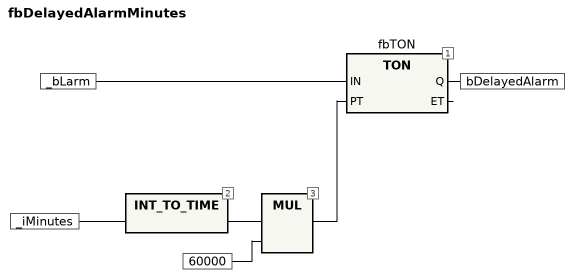
_CFC_ (* Continuous Function Chart, elements in execution order *)
#0 bDelayedAlarm <= #1.Q
#1 fbTON:TON(IN: _bLarm, PT: #3)
#2 INT_TO_TIME(_iMinutes)
#3 MUL(#2, 60000)
_END_CFC_
(* the same logic as Structured Text *)
bDelayedAlarm := fbTON.Q;
fbTON(IN := _bLarm, PT := _t13);
_t13 := INT_TO_TIME(_iMinutes) * 60000;
END_FUNCTION_BLOCK

(* POU xRIO_komfel/RIO_COM_L, CFC *)
PROGRAM RIO_COM_L
VAR

	State1 AT%I*:UINT;			(* Kommunikationsfel RIO1 *)
	State2 AT%I*:UINT;			(* Kommunikationsfel RIO2 *)
	State3 AT%I*:UINT;			(* Kommunikationsfel RIO3 *)
	State4 AT%I*:UINT;			(* Kommunikationsfel RIO4 *)
	State5 AT%I*:UINT;			(* Kommunikationsfel RIO5 *)

	KBusState1 AT%I*:UINT;			(* KBus/IO-fel  RIO1 *)
	KBusState2 AT%I*:UINT;			(* KBus/IO-fel  RIO2 *)
	KBusState3 AT%I*:UINT;			(* KBus/IO-fel  RIO3 *)
	KBusState4 AT%I*:UINT;			(* KBus/IO-fel  RIO4 *)
	KBusState5 AT%I*:UINT;			(* KBus/IO-fel  RIO5 *)

	Komfel1:BOOL;
	Komfel2:BOOL;
	Komfel3:BOOL;
	Komfel4:BOOL;
	Komfel5:BOOL;

	KBusfel1	:BOOL;
	KBusfel2	:BOOL;
	KBusfel3	:BOOL;
	KBusfel4	:BOOL;
	KBusfel5	:BOOL;

	KOMFELDELAY1: TON;
	KOMFELDELAY2: TON;
	KOMFELDELAY3: TON;
	KOMFELDELAY4: TON;
	KOMFELDELAY5: TON;
	IODELAY1: TON;
	IODELAY2: TON;
	IODELAY3: TON;
	IODELAY4: TON;
	IODELAY5: TON;
END_VAR
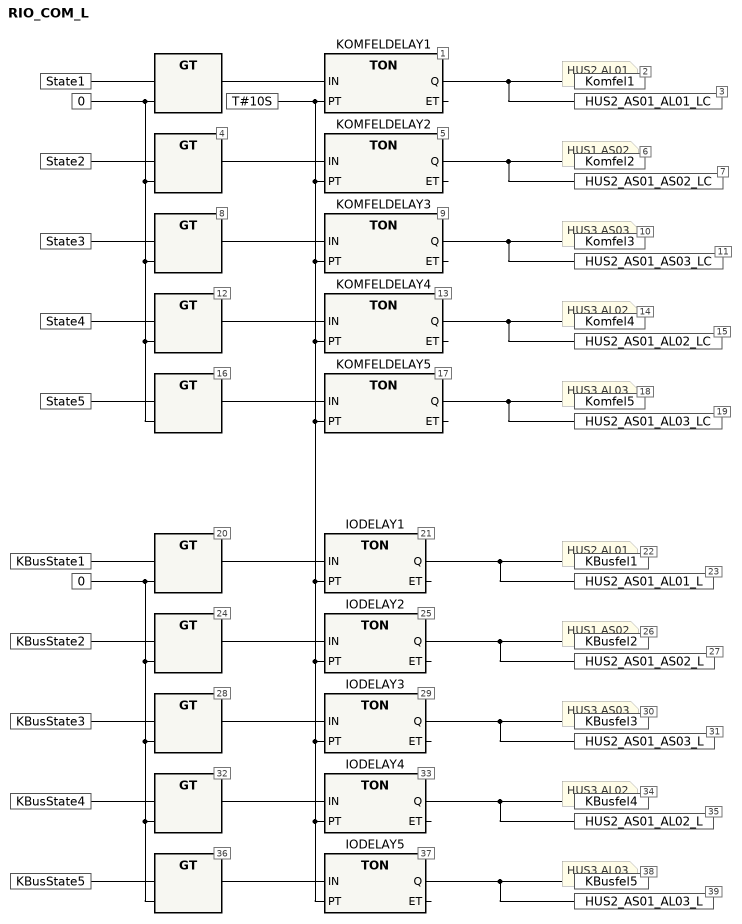
_CFC_ (* Continuous Function Chart, elements in execution order *)
(* HUS3 AL03 *)
(* HUS1 AS02 *)
(* HUS3 AL02 *)
(* HUS3 AS03 *)
(* HUS2 AL01 *)
(* HUS3 AL03 *)
(* HUS1 AS02 *)
(* HUS3 AL02 *)
(* HUS3 AS03 *)
(* HUS2 AL01 *)
#0 GT(State1, 0)
#1 KOMFELDELAY1:TON(IN: #0, PT: T#10S)
#2 Komfel1 <= #1.Q
#3 HUS2_AS01_AL01_LC <= #1.Q
#4 GT(State2, 0)
#5 KOMFELDELAY2:TON(IN: #4, PT: T#10S)
#6 Komfel2 <= #5.Q
#7 HUS2_AS01_AS02_LC <= #5.Q
#8 GT(State3, 0)
#9 KOMFELDELAY3:TON(IN: #8, PT: T#10S)
#10 Komfel3 <= #9.Q
#11 HUS2_AS01_AS03_LC <= #9.Q
#12 GT(State4, 0)
#13 KOMFELDELAY4:TON(IN: #12, PT: T#10S)
#14 Komfel4 <= #13.Q
#15 HUS2_AS01_AL02_LC <= #13.Q
#16 GT(State5, 0)
#17 KOMFELDELAY5:TON(IN: #16, PT: T#10S)
#18 Komfel5 <= #17.Q
#19 HUS2_AS01_AL03_LC <= #17.Q
#20 GT(KBusState1, 0)
#21 IODELAY1:TON(IN: #20, PT: T#10S)
#22 KBusfel1 <= #21.Q
#23 HUS2_AS01_AL01_L <= #21.Q
#24 GT(KBusState2, 0)
#25 IODELAY2:TON(IN: #24, PT: T#10S)
#26 KBusfel2 <= #25.Q
#27 HUS2_AS01_AS02_L <= #25.Q
#28 GT(KBusState3, 0)
#29 IODELAY3:TON(IN: #28, PT: T#10S)
#30 KBusfel3 <= #29.Q
#31 HUS2_AS01_AS03_L <= #29.Q
#32 GT(KBusState4, 0)
#33 IODELAY4:TON(IN: #32, PT: T#10S)
#34 KBusfel4 <= #33.Q
#35 HUS2_AS01_AL02_L <= #33.Q
#36 GT(KBusState5, 0)
#37 IODELAY5:TON(IN: #36, PT: T#10S)
#38 KBusfel5 <= #37.Q
#39 HUS2_AS01_AL03_L <= #37.Q
_END_CFC_
(* the same logic as Structured Text *)
(* HUS3 AL03 *)
(* HUS1 AS02 *)
(* HUS3 AL02 *)
(* HUS3 AS03 *)
(* HUS2 AL01 *)
(* HUS3 AL03 *)
(* HUS1 AS02 *)
(* HUS3 AL02 *)
(* HUS3 AS03 *)
(* HUS2 AL01 *)
KOMFELDELAY1(IN := State1 > 0, PT := T#10S);
Komfel1 := KOMFELDELAY1.Q;
HUS2_AS01_AL01_LC := KOMFELDELAY1.Q;
KOMFELDELAY2(IN := State2 > 0, PT := T#10S);
Komfel2 := KOMFELDELAY2.Q;
HUS2_AS01_AS02_LC := KOMFELDELAY2.Q;
KOMFELDELAY3(IN := State3 > 0, PT := T#10S);
Komfel3 := KOMFELDELAY3.Q;
HUS2_AS01_AS03_LC := KOMFELDELAY3.Q;
KOMFELDELAY4(IN := State4 > 0, PT := T#10S);
Komfel4 := KOMFELDELAY4.Q;
HUS2_AS01_AL02_LC := KOMFELDELAY4.Q;
KOMFELDELAY5(IN := State5 > 0, PT := T#10S);
Komfel5 := KOMFELDELAY5.Q;
HUS2_AS01_AL03_LC := KOMFELDELAY5.Q;
IODELAY1(IN := KBusState1 > 0, PT := T#10S);
KBusfel1 := IODELAY1.Q;
HUS2_AS01_AL01_L := IODELAY1.Q;
IODELAY2(IN := KBusState2 > 0, PT := T#10S);
KBusfel2 := IODELAY2.Q;
HUS2_AS01_AS02_L := IODELAY2.Q;
IODELAY3(IN := KBusState3 > 0, PT := T#10S);
KBusfel3 := IODELAY3.Q;
HUS2_AS01_AS03_L := IODELAY3.Q;
IODELAY4(IN := KBusState4 > 0, PT := T#10S);
KBusfel4 := IODELAY4.Q;
HUS2_AS01_AL02_L := IODELAY4.Q;
IODELAY5(IN := KBusState5 > 0, PT := T#10S);
KBusfel5 := IODELAY5.Q;
HUS2_AS01_AL03_L := IODELAY5.Q;
END_PROGRAM

(* POU _IOs_Uppdelat_per_skåp/HUS1_AS02/_IO/HUS1_AS02_IO_MAIN, CFC *)
PROGRAM HUS1_AS02_IO_MAIN
VAR
END_VAR
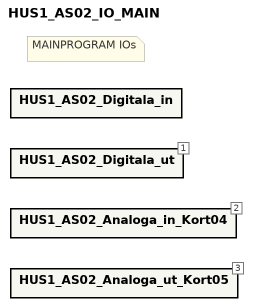
_CFC_ (* Continuous Function Chart, elements in execution order *)
(* MAINPROGRAM IOs *)
#0 HUS1_AS02_Digitala_in()
#1 HUS1_AS02_Digitala_ut()
#2 HUS1_AS02_Analoga_in_Kort04()
#3 HUS1_AS02_Analoga_ut_Kort05()
_END_CFC_
(* the same logic as Structured Text *)
(* MAINPROGRAM IOs *)
HUS1_AS02_Digitala_in();
HUS1_AS02_Digitala_ut();
HUS1_AS02_Analoga_in_Kort04();
HUS1_AS02_Analoga_ut_Kort05();
END_PROGRAM

(* POU _IOs_Uppdelat_per_skåp/HUS1_AS02/_IO/HUS1_AS02_Digitala_in, CFC *)
PROGRAM HUS1_AS02_Digitala_in

VAR


END_VAR
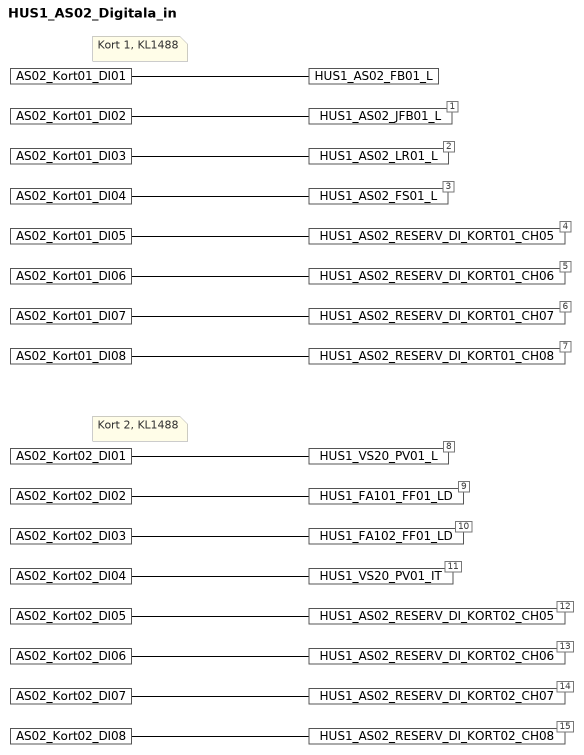
_CFC_ (* Continuous Function Chart, elements in execution order *)
(* Kort 1, KL1488 *)
(* Kort 2, KL1488 *)
#0 HUS1_AS02_FB01_L <= AS02_Kort01_DI01
#1 HUS1_AS02_JFB01_L <= AS02_Kort01_DI02
#2 HUS1_AS02_LR01_L <= AS02_Kort01_DI03
#3 HUS1_AS02_FS01_L <= AS02_Kort01_DI04
#4 HUS1_AS02_RESERV_DI_KORT01_CH05 <= AS02_Kort01_DI05
#5 HUS1_AS02_RESERV_DI_KORT01_CH06 <= AS02_Kort01_DI06
#6 HUS1_AS02_RESERV_DI_KORT01_CH07 <= AS02_Kort01_DI07
#7 HUS1_AS02_RESERV_DI_KORT01_CH08 <= AS02_Kort01_DI08
#8 HUS1_VS20_PV01_L <= AS02_Kort02_DI01
#9 HUS1_FA101_FF01_LD <= AS02_Kort02_DI02
#10 HUS1_FA102_FF01_LD <= AS02_Kort02_DI03
#11 HUS1_VS20_PV01_IT <= AS02_Kort02_DI04
#12 HUS1_AS02_RESERV_DI_KORT02_CH05 <= AS02_Kort02_DI05
#13 HUS1_AS02_RESERV_DI_KORT02_CH06 <= AS02_Kort02_DI06
#14 HUS1_AS02_RESERV_DI_KORT02_CH07 <= AS02_Kort02_DI07
#15 HUS1_AS02_RESERV_DI_KORT02_CH08 <= AS02_Kort02_DI08
_END_CFC_
(* the same logic as Structured Text *)
(* Kort 1, KL1488 *)
(* Kort 2, KL1488 *)
HUS1_AS02_FB01_L := AS02_Kort01_DI01;
HUS1_AS02_JFB01_L := AS02_Kort01_DI02;
HUS1_AS02_LR01_L := AS02_Kort01_DI03;
HUS1_AS02_FS01_L := AS02_Kort01_DI04;
HUS1_AS02_RESERV_DI_KORT01_CH05 := AS02_Kort01_DI05;
HUS1_AS02_RESERV_DI_KORT01_CH06 := AS02_Kort01_DI06;
HUS1_AS02_RESERV_DI_KORT01_CH07 := AS02_Kort01_DI07;
HUS1_AS02_RESERV_DI_KORT01_CH08 := AS02_Kort01_DI08;
HUS1_VS20_PV01_L := AS02_Kort02_DI01;
HUS1_FA101_FF01_LD := AS02_Kort02_DI02;
HUS1_FA102_FF01_LD := AS02_Kort02_DI03;
HUS1_VS20_PV01_IT := AS02_Kort02_DI04;
HUS1_AS02_RESERV_DI_KORT02_CH05 := AS02_Kort02_DI05;
HUS1_AS02_RESERV_DI_KORT02_CH06 := AS02_Kort02_DI06;
HUS1_AS02_RESERV_DI_KORT02_CH07 := AS02_Kort02_DI07;
HUS1_AS02_RESERV_DI_KORT02_CH08 := AS02_Kort02_DI08;
END_PROGRAM

(* POU _IOs_Uppdelat_per_skåp/HUS1_AS02/_IO/HUS1_AS02_Digitala_ut, CFC *)
PROGRAM HUS1_AS02_Digitala_ut


VAR
	HUS1_Kort03_DU01: BOOL;
	HUS1_Kort03_DU02: BOOL;
	HUS1_Kort03_DU03: BOOL;
	HUS1_HUS1_RESERV_DU_KORT03_CH04: BOOL;
	HUS1_Kort03_DU04: BOOL;
END_VAR
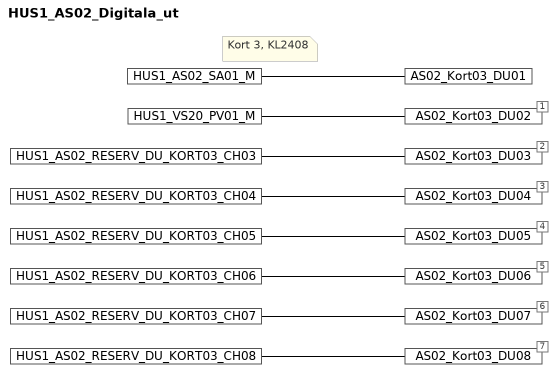
_CFC_ (* Continuous Function Chart, elements in execution order *)
(* Kort 3, KL2408 *)
#0 AS02_Kort03_DU01 <= HUS1_AS02_SA01_M
#1 AS02_Kort03_DU02 <= HUS1_VS20_PV01_M
#2 AS02_Kort03_DU03 <= HUS1_AS02_RESERV_DU_KORT03_CH03
#3 AS02_Kort03_DU04 <= HUS1_AS02_RESERV_DU_KORT03_CH04
#4 AS02_Kort03_DU05 <= HUS1_AS02_RESERV_DU_KORT03_CH05
#5 AS02_Kort03_DU06 <= HUS1_AS02_RESERV_DU_KORT03_CH06
#6 AS02_Kort03_DU07 <= HUS1_AS02_RESERV_DU_KORT03_CH07
#7 AS02_Kort03_DU08 <= HUS1_AS02_RESERV_DU_KORT03_CH08
_END_CFC_
(* the same logic as Structured Text *)
(* Kort 3, KL2408 *)
AS02_Kort03_DU01 := HUS1_AS02_SA01_M;
AS02_Kort03_DU02 := HUS1_VS20_PV01_M;
AS02_Kort03_DU03 := HUS1_AS02_RESERV_DU_KORT03_CH03;
AS02_Kort03_DU04 := HUS1_AS02_RESERV_DU_KORT03_CH04;
AS02_Kort03_DU05 := HUS1_AS02_RESERV_DU_KORT03_CH05;
AS02_Kort03_DU06 := HUS1_AS02_RESERV_DU_KORT03_CH06;
AS02_Kort03_DU07 := HUS1_AS02_RESERV_DU_KORT03_CH07;
AS02_Kort03_DU08 := HUS1_AS02_RESERV_DU_KORT03_CH08;
END_PROGRAM

(* POU _IOs_Uppdelat_per_skåp/HUS1_AS02/_IO/ANALOGA IN/Kort04/HUS1_AS02_Analoga_in_Kort04, CFC *)
PROGRAM HUS1_AS02_Analoga_in_Kort04
VAR
	bLG01: BOOL;
	bLG02: BOOL;
	bLG03: BOOL;
	bLG04: BOOL;
	bLG05: BOOL;
	bLG06: BOOL;
	bLG07: BOOL;
	bLG08: BOOL;

(*TEMP*)
	FT1:INT;
	LG_FL1:INT;
	FT2:INT;
	LG_FL2:INT;
	FT3:INT;
	LG_FL3:INT;
	FT4:INT;
	LG_FL4:INT;
	FT5:INT;
	LG_FL5:INT;
	FT6:INT;
	LG_FL6:INT;
	FT7:INT;
	LG_FL7:INT;
	FT8:INT;
	LG_FL8:INT;

END_VAR
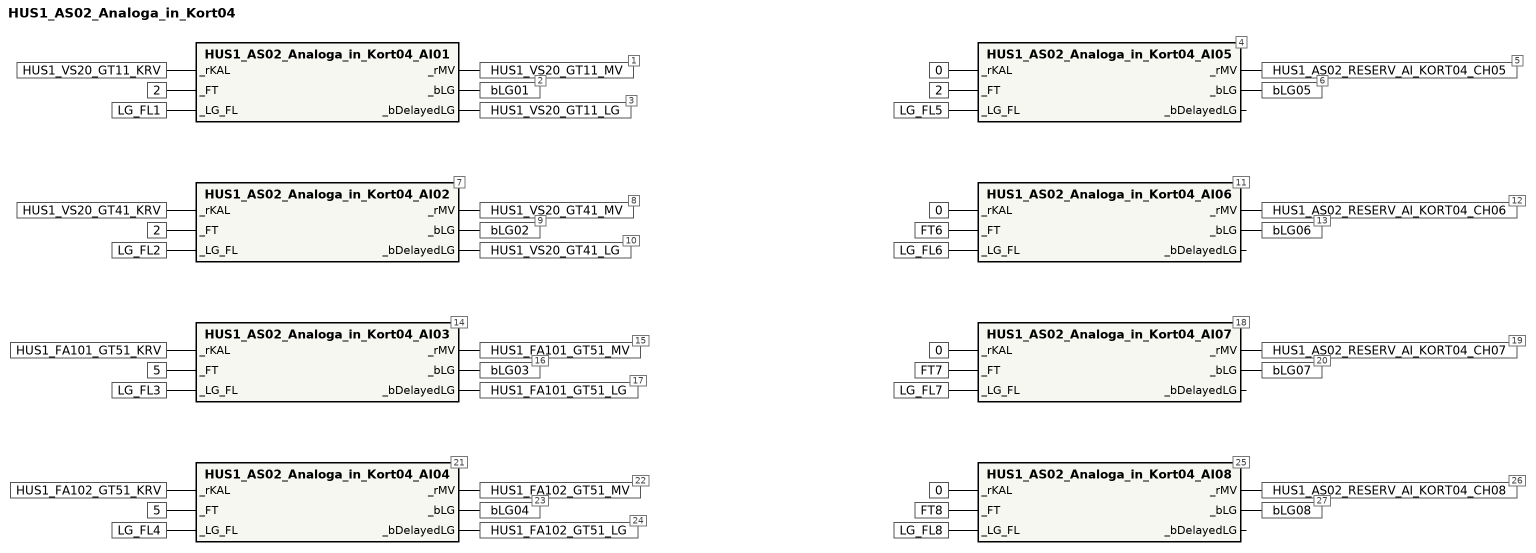
_CFC_ (* Continuous Function Chart, elements in execution order *)
#0 HUS1_AS02_Analoga_in_Kort04_AI01(_rKAL: HUS1_VS20_GT11_KRV, _FT: 2, _LG_FL: LG_FL1)
#1 HUS1_VS20_GT11_MV <= #0._rMV
#2 bLG01 <= #0._bLG
#3 HUS1_VS20_GT11_LG <= #0._bDelayedLG
#4 HUS1_AS02_Analoga_in_Kort04_AI05(_rKAL: 0, _FT: 2, _LG_FL: LG_FL5)
#5 HUS1_AS02_RESERV_AI_KORT04_CH05 <= #4._rMV
#6 bLG05 <= #4._bLG
#7 HUS1_AS02_Analoga_in_Kort04_AI02(_rKAL: HUS1_VS20_GT41_KRV, _FT: 2, _LG_FL: LG_FL2)
#8 HUS1_VS20_GT41_MV <= #7._rMV
#9 bLG02 <= #7._bLG
#10 HUS1_VS20_GT41_LG <= #7._bDelayedLG
#11 HUS1_AS02_Analoga_in_Kort04_AI06(_rKAL: 0, _FT: FT6, _LG_FL: LG_FL6)
#12 HUS1_AS02_RESERV_AI_KORT04_CH06 <= #11._rMV
#13 bLG06 <= #11._bLG
#14 HUS1_AS02_Analoga_in_Kort04_AI03(_rKAL: HUS1_FA101_GT51_KRV, _FT: 5, _LG_FL: LG_FL3)
#15 HUS1_FA101_GT51_MV <= #14._rMV
#16 bLG03 <= #14._bLG
#17 HUS1_FA101_GT51_LG <= #14._bDelayedLG
#18 HUS1_AS02_Analoga_in_Kort04_AI07(_rKAL: 0, _FT: FT7, _LG_FL: LG_FL7)
#19 HUS1_AS02_RESERV_AI_KORT04_CH07 <= #18._rMV
#20 bLG07 <= #18._bLG
#21 HUS1_AS02_Analoga_in_Kort04_AI04(_rKAL: HUS1_FA102_GT51_KRV, _FT: 5, _LG_FL: LG_FL4)
#22 HUS1_FA102_GT51_MV <= #21._rMV
#23 bLG04 <= #21._bLG
#24 HUS1_FA102_GT51_LG <= #21._bDelayedLG
#25 HUS1_AS02_Analoga_in_Kort04_AI08(_rKAL: 0, _FT: FT8, _LG_FL: LG_FL8)
#26 HUS1_AS02_RESERV_AI_KORT04_CH08 <= #25._rMV
#27 bLG08 <= #25._bLG
_END_CFC_
(* the same logic as Structured Text *)
HUS1_AS02_Analoga_in_Kort04_AI01(_rKAL := HUS1_VS20_GT11_KRV, _FT := 2, _LG_FL := LG_FL1);
HUS1_VS20_GT11_MV := HUS1_AS02_Analoga_in_Kort04_AI01._rMV;
bLG01 := HUS1_AS02_Analoga_in_Kort04_AI01._bLG;
HUS1_VS20_GT11_LG := HUS1_AS02_Analoga_in_Kort04_AI01._bDelayedLG;
HUS1_AS02_Analoga_in_Kort04_AI05(_rKAL := 0, _FT := 2, _LG_FL := LG_FL5);
HUS1_AS02_RESERV_AI_KORT04_CH05 := HUS1_AS02_Analoga_in_Kort04_AI05._rMV;
bLG05 := HUS1_AS02_Analoga_in_Kort04_AI05._bLG;
HUS1_AS02_Analoga_in_Kort04_AI02(_rKAL := HUS1_VS20_GT41_KRV, _FT := 2, _LG_FL := LG_FL2);
HUS1_VS20_GT41_MV := HUS1_AS02_Analoga_in_Kort04_AI02._rMV;
bLG02 := HUS1_AS02_Analoga_in_Kort04_AI02._bLG;
HUS1_VS20_GT41_LG := HUS1_AS02_Analoga_in_Kort04_AI02._bDelayedLG;
HUS1_AS02_Analoga_in_Kort04_AI06(_rKAL := 0, _FT := FT6, _LG_FL := LG_FL6);
HUS1_AS02_RESERV_AI_KORT04_CH06 := HUS1_AS02_Analoga_in_Kort04_AI06._rMV;
bLG06 := HUS1_AS02_Analoga_in_Kort04_AI06._bLG;
HUS1_AS02_Analoga_in_Kort04_AI03(_rKAL := HUS1_FA101_GT51_KRV, _FT := 5, _LG_FL := LG_FL3);
HUS1_FA101_GT51_MV := HUS1_AS02_Analoga_in_Kort04_AI03._rMV;
bLG03 := HUS1_AS02_Analoga_in_Kort04_AI03._bLG;
HUS1_FA101_GT51_LG := HUS1_AS02_Analoga_in_Kort04_AI03._bDelayedLG;
HUS1_AS02_Analoga_in_Kort04_AI07(_rKAL := 0, _FT := FT7, _LG_FL := LG_FL7);
HUS1_AS02_RESERV_AI_KORT04_CH07 := HUS1_AS02_Analoga_in_Kort04_AI07._rMV;
bLG07 := HUS1_AS02_Analoga_in_Kort04_AI07._bLG;
HUS1_AS02_Analoga_in_Kort04_AI04(_rKAL := HUS1_FA102_GT51_KRV, _FT := 5, _LG_FL := LG_FL4);
HUS1_FA102_GT51_MV := HUS1_AS02_Analoga_in_Kort04_AI04._rMV;
bLG04 := HUS1_AS02_Analoga_in_Kort04_AI04._bLG;
HUS1_FA102_GT51_LG := HUS1_AS02_Analoga_in_Kort04_AI04._bDelayedLG;
HUS1_AS02_Analoga_in_Kort04_AI08(_rKAL := 0, _FT := FT8, _LG_FL := LG_FL8);
HUS1_AS02_RESERV_AI_KORT04_CH08 := HUS1_AS02_Analoga_in_Kort04_AI08._rMV;
bLG08 := HUS1_AS02_Analoga_in_Kort04_AI08._bLG;
END_PROGRAM

(* POU _IOs_Uppdelat_per_skåp/HUS1_AS02/_IO/ANALOGA IN/Kort04/HUS1_AS02_Analoga_in_Kort04_AI01, FAI *)
PROGRAM HUS1_AS02_Analoga_in_Kort04_AI01
(*#####################################   Temperature Sensor Ex2   ################################################################*)
VAR
	(*===========================Configuration of terminal==========================================*)
	fbConfigureKL32xx					:FB_HVACConfigureKL32xx;
	_byCtrlKL32xx                         			AT %Q*: BYTE;
	_iDataOutKL32xx                       		AT %Q*: INT;
	_iDataInKL32xx 					AT%I*:INT;(* Raw Value from the Terminal *)
	_byStatusKL32xx 			AT%I*:BYTE;(* Statusbyte from Terminal *)

	_bScanSensor              					: BOOL;
	_tTimeOut                 					: TIME := T#5s;
	_bSetSensor               					: BOOL;
	bReady                               				: BOOL;
	byOutStatus                          			: BYTE;
	iOutDataIn                           				: INT;
	_eBusTerminalKL32xx                   		: E_HVACBusTerminal_KL32xx;
	_eStatusScanSensorType                	: E_HVACSensorType;
	_bErrorGeneral                        			: BOOL;
	_byError                              				: BYTE;
	_bErrorCommunication                  		: BOOL;
	_bErrorBusTerminalNotSupported   	: BOOL;
	_bErrorSensorType                     		: BOOL;
	_bErrorScanSensor                     		: BOOL;
	(*========================================================================================*)

	_bReset_Local					:BOOL;
	_bSetDefaultTempSens			:BOOL;

	(*========================================================================================*)
	FBHVACTemperatureSensor: FB_HVACTemperatureSensor;
	eDataSecurityType					: E_HVACDataSecurityType:=1;
	bSetDefault								:BOOL;
	iRawValue								:INT;
	byStatusRawValue						:BYTE;
	bEnableLimitCtrl							:BOOL;
	bReset									:BOOL;
	bErrorGeneral					:BOOL;
	byError							:BYTE;
	bErrorShortCircuit				:BOOL;
	bErrorBrokenSensor				:BOOL;
	bErrorHighLimit					:BOOL;
	bErrorLowLimit					:BOOL;
	bErrorCycleTime					:BOOL;
	bInvalidParameter				:BOOL;
	rOffset									:REAL;
	rHighLimit								:REAL;
	rLowLimit								:REAL;
	rReplacementValue						:REAL;
	tFilterTime								:TIME;
	eTemperatureSensorMode				:E_HVACTemperatureSensorMode:=2;
	fbAlarmD: fbDelayedAlarmMinutes;

END_VAR

VAR_INPUT
	_rKAL						: REAL;	(*Kalibrering*)
	_FT						:INT;		(*Filtertid*)
	_LG_FL					:INT;		(* Larmfördröjning givarfel *)
END_VAR

VAR_OUTPUT
	_rMV						:REAL;		(* Mätvärde *)
	_bLG						:BOOL; 	(*Givarfel*)
	_bDelayedLG				:BOOL;	(* Fördröjt givarfel *)
END_VAR
(* body not read: cfc101 *)
END_PROGRAM

(* POU _IOs_Uppdelat_per_skåp/HUS1_AS02/_IO/ANALOGA IN/Kort04/HUS1_AS02_Analoga_in_Kort04_AI05, FAI *)
PROGRAM HUS1_AS02_Analoga_in_Kort04_AI05
(*#####################################   Temperature Sensor Ex2   ################################################################*)
VAR
	(*===========================Configuration of terminal==========================================*)
	fbConfigureKL32xx					:FB_HVACConfigureKL32xx;
	_byCtrlKL32xx                         			AT %Q*: BYTE;
	_iDataOutKL32xx                       		AT %Q*: INT;
	_iDataInKL32xx 					AT%I*:INT;(* Raw Value from the Terminal *)
	_byStatusKL32xx 			AT%I*:BYTE;(* Statusbyte from Terminal *)

	_bScanSensor              					: BOOL;
	_tTimeOut                 					: TIME := T#5s;
	_bSetSensor               					: BOOL;
	bReady                               				: BOOL;
	byOutStatus                          			: BYTE;
	iOutDataIn                           				: INT;
	_eBusTerminalKL32xx                   		: E_HVACBusTerminal_KL32xx;
	_eStatusScanSensorType                	: E_HVACSensorType;
	_bErrorGeneral                        			: BOOL;
	_byError                              				: BYTE;
	_bErrorCommunication                  		: BOOL;
	_bErrorBusTerminalNotSupported   	: BOOL;
	_bErrorSensorType                     		: BOOL;
	_bErrorScanSensor                     		: BOOL;
	(*========================================================================================*)

	_bReset_Local					:BOOL;
	_bSetDefaultTempSens			:BOOL;

	(*========================================================================================*)
	FBHVACTemperatureSensor: FB_HVACTemperatureSensor;
	eDataSecurityType					: E_HVACDataSecurityType:=1;
	bSetDefault								:BOOL;
	iRawValue								:INT;
	byStatusRawValue						:BYTE;
	bEnableLimitCtrl							:BOOL;
	bReset									:BOOL;
	bErrorGeneral					:BOOL;
	byError							:BYTE;
	bErrorShortCircuit				:BOOL;
	bErrorBrokenSensor				:BOOL;
	bErrorHighLimit					:BOOL;
	bErrorLowLimit					:BOOL;
	bErrorCycleTime					:BOOL;
	bInvalidParameter				:BOOL;
	rOffset									:REAL;
	rHighLimit								:REAL;
	rLowLimit								:REAL;
	rReplacementValue						:REAL;
	tFilterTime								:TIME;
	eTemperatureSensorMode				:E_HVACTemperatureSensorMode:=2;
	fbAlarmD: fbDelayedAlarmMinutes;

END_VAR

VAR_INPUT
	_rKAL						: REAL;	(*Kalibrering*)
	_FT						:INT;		(*Filtertid*)
	_LG_FL					:INT;		(* Larmfördröjning givarfel *)
END_VAR

VAR_OUTPUT
	_rMV						:REAL;		(* Mätvärde *)
	_bLG						:BOOL; 	(*Givarfel*)
	_bDelayedLG				:BOOL;	(* Fördröjt givarfel *)
END_VAR
(* body not read: cfc101 *)
END_PROGRAM

(* POU _IOs_Uppdelat_per_skåp/HUS1_AS02/_IO/ANALOGA IN/Kort04/HUS1_AS02_Analoga_in_Kort04_AI02, FAI *)
PROGRAM HUS1_AS02_Analoga_in_Kort04_AI02
(*#####################################   Temperature Sensor Ex2   ################################################################*)
VAR
	(*===========================Configuration of terminal==========================================*)
	fbConfigureKL32xx					:FB_HVACConfigureKL32xx;
	_byCtrlKL32xx                         			AT %Q*: BYTE;
	_iDataOutKL32xx                       		AT %Q*: INT;
	_iDataInKL32xx 					AT%I*:INT;(* Raw Value from the Terminal *)
	_byStatusKL32xx 			AT%I*:BYTE;(* Statusbyte from Terminal *)

	_bScanSensor              					: BOOL;
	_tTimeOut                 					: TIME := T#5s;
	_bSetSensor               					: BOOL;
	bReady                               				: BOOL;
	byOutStatus                          			: BYTE;
	iOutDataIn                           				: INT;
	_eBusTerminalKL32xx                   		: E_HVACBusTerminal_KL32xx;
	_eStatusScanSensorType                	: E_HVACSensorType;
	_bErrorGeneral                        			: BOOL;
	_byError                              				: BYTE;
	_bErrorCommunication                  		: BOOL;
	_bErrorBusTerminalNotSupported   	: BOOL;
	_bErrorSensorType                     		: BOOL;
	_bErrorScanSensor                     		: BOOL;
	(*========================================================================================*)

	_bReset_Local					:BOOL;
	_bSetDefaultTempSens			:BOOL;

	(*========================================================================================*)
	FBHVACTemperatureSensor: FB_HVACTemperatureSensor;
	eDataSecurityType					: E_HVACDataSecurityType:=1;
	bSetDefault								:BOOL;
	iRawValue								:INT;
	byStatusRawValue						:BYTE;
	bEnableLimitCtrl							:BOOL;
	bReset									:BOOL;
	bErrorGeneral					:BOOL;
	byError							:BYTE;
	bErrorShortCircuit				:BOOL;
	bErrorBrokenSensor				:BOOL;
	bErrorHighLimit					:BOOL;
	bErrorLowLimit					:BOOL;
	bErrorCycleTime					:BOOL;
	bInvalidParameter				:BOOL;
	rOffset									:REAL;
	rHighLimit								:REAL;
	rLowLimit								:REAL;
	rReplacementValue						:REAL;
	tFilterTime								:TIME;
	eTemperatureSensorMode				:E_HVACTemperatureSensorMode:=2;
	fbAlarmD: fbDelayedAlarmMinutes;

END_VAR

VAR_INPUT
	_rKAL						: REAL;	(*Kalibrering*)
	_FT						:INT;		(*Filtertid*)
	_LG_FL					:INT;		(* Larmfördröjning givarfel *)
END_VAR

VAR_OUTPUT
	_rMV						:REAL;		(* Mätvärde *)
	_bLG						:BOOL; 	(*Givarfel*)
	_bDelayedLG				:BOOL;	(* Fördröjt givarfel *)
END_VAR
(* body not read: cfc101 *)
END_PROGRAM

(* POU _IOs_Uppdelat_per_skåp/HUS1_AS02/_IO/ANALOGA IN/Kort04/HUS1_AS02_Analoga_in_Kort04_AI06, FAI *)
PROGRAM HUS1_AS02_Analoga_in_Kort04_AI06
(*#####################################   Temperature Sensor Ex2   ################################################################*)
VAR
	(*===========================Configuration of terminal==========================================*)
	fbConfigureKL32xx					:FB_HVACConfigureKL32xx;
	_byCtrlKL32xx                         			AT %Q*: BYTE;
	_iDataOutKL32xx                       		AT %Q*: INT;
	_iDataInKL32xx 					AT%I*:INT;(* Raw Value from the Terminal *)
	_byStatusKL32xx 			AT%I*:BYTE;(* Statusbyte from Terminal *)

	_bScanSensor              					: BOOL;
	_tTimeOut                 					: TIME := T#5s;
	_bSetSensor               					: BOOL;
	bReady                               				: BOOL;
	byOutStatus                          			: BYTE;
	iOutDataIn                           				: INT;
	_eBusTerminalKL32xx                   		: E_HVACBusTerminal_KL32xx;
	_eStatusScanSensorType                	: E_HVACSensorType;
	_bErrorGeneral                        			: BOOL;
	_byError                              				: BYTE;
	_bErrorCommunication                  		: BOOL;
	_bErrorBusTerminalNotSupported   	: BOOL;
	_bErrorSensorType                     		: BOOL;
	_bErrorScanSensor                     		: BOOL;
	(*========================================================================================*)

	_bReset_Local					:BOOL;
	_bSetDefaultTempSens			:BOOL;

	(*========================================================================================*)
	FBHVACTemperatureSensor: FB_HVACTemperatureSensor;
	eDataSecurityType					: E_HVACDataSecurityType:=1;
	bSetDefault								:BOOL;
	iRawValue								:INT;
	byStatusRawValue						:BYTE;
	bEnableLimitCtrl							:BOOL;
	bReset									:BOOL;
	bErrorGeneral					:BOOL;
	byError							:BYTE;
	bErrorShortCircuit				:BOOL;
	bErrorBrokenSensor				:BOOL;
	bErrorHighLimit					:BOOL;
	bErrorLowLimit					:BOOL;
	bErrorCycleTime					:BOOL;
	bInvalidParameter				:BOOL;
	rOffset									:REAL;
	rHighLimit								:REAL;
	rLowLimit								:REAL;
	rReplacementValue						:REAL;
	tFilterTime								:TIME;
	eTemperatureSensorMode				:E_HVACTemperatureSensorMode:=2;
	fbAlarmD: fbDelayedAlarmMinutes;

END_VAR

VAR_INPUT
	_rKAL						: REAL;	(*Kalibrering*)
	_FT						:INT;		(*Filtertid*)
	_LG_FL					:INT;		(* Larmfördröjning givarfel *)
END_VAR

VAR_OUTPUT
	_rMV						:REAL;		(* Mätvärde *)
	_bLG						:BOOL; 	(*Givarfel*)
	_bDelayedLG				:BOOL;	(* Fördröjt givarfel *)
END_VAR
(* body not read: cfc101 *)
END_PROGRAM

(* POU _IOs_Uppdelat_per_skåp/HUS1_AS02/_IO/ANALOGA IN/Kort04/HUS1_AS02_Analoga_in_Kort04_AI03, FAI *)
PROGRAM HUS1_AS02_Analoga_in_Kort04_AI03
(*#####################################   Temperature Sensor Ex2   ################################################################*)
VAR
	(*===========================Configuration of terminal==========================================*)
	fbConfigureKL32xx					:FB_HVACConfigureKL32xx;
	_byCtrlKL32xx                         			AT %Q*: BYTE;
	_iDataOutKL32xx                       		AT %Q*: INT;
	_iDataInKL32xx 					AT%I*:INT;(* Raw Value from the Terminal *)
	_byStatusKL32xx 			AT%I*:BYTE;(* Statusbyte from Terminal *)

	_bScanSensor              					: BOOL;
	_tTimeOut                 					: TIME := T#5s;
	_bSetSensor               					: BOOL;
	bReady                               				: BOOL;
	byOutStatus                          			: BYTE;
	iOutDataIn                           				: INT;
	_eBusTerminalKL32xx                   		: E_HVACBusTerminal_KL32xx;
	_eStatusScanSensorType                	: E_HVACSensorType;
	_bErrorGeneral                        			: BOOL;
	_byError                              				: BYTE;
	_bErrorCommunication                  		: BOOL;
	_bErrorBusTerminalNotSupported   	: BOOL;
	_bErrorSensorType                     		: BOOL;
	_bErrorScanSensor                     		: BOOL;
	(*========================================================================================*)

	_bReset_Local					:BOOL;
	_bSetDefaultTempSens			:BOOL;

	(*========================================================================================*)
	FBHVACTemperatureSensor: FB_HVACTemperatureSensor;
	eDataSecurityType					: E_HVACDataSecurityType:=1;
	bSetDefault								:BOOL;
	iRawValue								:INT;
	byStatusRawValue						:BYTE;
	bEnableLimitCtrl							:BOOL;
	bReset									:BOOL;
	bErrorGeneral					:BOOL;
	byError							:BYTE;
	bErrorShortCircuit				:BOOL;
	bErrorBrokenSensor				:BOOL;
	bErrorHighLimit					:BOOL;
	bErrorLowLimit					:BOOL;
	bErrorCycleTime					:BOOL;
	bInvalidParameter				:BOOL;
	rOffset									:REAL;
	rHighLimit								:REAL;
	rLowLimit								:REAL;
	rReplacementValue						:REAL;
	tFilterTime								:TIME;
	eTemperatureSensorMode				:E_HVACTemperatureSensorMode:=2;
	fbAlarmD: fbDelayedAlarmMinutes;

END_VAR

VAR_INPUT
	_rKAL						: REAL;	(*Kalibrering*)
	_FT						:INT;		(*Filtertid*)
	_LG_FL					:INT;		(* Larmfördröjning givarfel *)
END_VAR

VAR_OUTPUT
	_rMV						:REAL;		(* Mätvärde *)
	_bLG						:BOOL; 	(*Givarfel*)
	_bDelayedLG				:BOOL;	(* Fördröjt givarfel *)
END_VAR
(* body not read: cfc101 *)
END_PROGRAM

(* POU _IOs_Uppdelat_per_skåp/HUS1_AS02/_IO/ANALOGA IN/Kort04/HUS1_AS02_Analoga_in_Kort04_AI07, FAI *)
PROGRAM HUS1_AS02_Analoga_in_Kort04_AI07
(*#####################################   Temperature Sensor Ex2   ################################################################*)
VAR
	(*===========================Configuration of terminal==========================================*)
	fbConfigureKL32xx					:FB_HVACConfigureKL32xx;
	_byCtrlKL32xx                         			AT %Q*: BYTE;
	_iDataOutKL32xx                       		AT %Q*: INT;
	_iDataInKL32xx 					AT%I*:INT;(* Raw Value from the Terminal *)
	_byStatusKL32xx 			AT%I*:BYTE;(* Statusbyte from Terminal *)

	_bScanSensor              					: BOOL;
	_tTimeOut                 					: TIME := T#5s;
	_bSetSensor               					: BOOL;
	bReady                               				: BOOL;
	byOutStatus                          			: BYTE;
	iOutDataIn                           				: INT;
	_eBusTerminalKL32xx                   		: E_HVACBusTerminal_KL32xx;
	_eStatusScanSensorType                	: E_HVACSensorType;
	_bErrorGeneral                        			: BOOL;
	_byError                              				: BYTE;
	_bErrorCommunication                  		: BOOL;
	_bErrorBusTerminalNotSupported   	: BOOL;
	_bErrorSensorType                     		: BOOL;
	_bErrorScanSensor                     		: BOOL;
	(*========================================================================================*)

	_bReset_Local					:BOOL;
	_bSetDefaultTempSens			:BOOL;

	(*========================================================================================*)
	FBHVACTemperatureSensor: FB_HVACTemperatureSensor;
	eDataSecurityType					: E_HVACDataSecurityType:=1;
	bSetDefault								:BOOL;
	iRawValue								:INT;
	byStatusRawValue						:BYTE;
	bEnableLimitCtrl							:BOOL;
	bReset									:BOOL;
	bErrorGeneral					:BOOL;
	byError							:BYTE;
	bErrorShortCircuit				:BOOL;
	bErrorBrokenSensor				:BOOL;
	bErrorHighLimit					:BOOL;
	bErrorLowLimit					:BOOL;
	bErrorCycleTime					:BOOL;
	bInvalidParameter				:BOOL;
	rOffset									:REAL;
	rHighLimit								:REAL;
	rLowLimit								:REAL;
	rReplacementValue						:REAL;
	tFilterTime								:TIME;
	eTemperatureSensorMode				:E_HVACTemperatureSensorMode:=2;
	fbAlarmD: fbDelayedAlarmMinutes;

END_VAR

VAR_INPUT
	_rKAL						: REAL;	(*Kalibrering*)
	_FT						:INT;		(*Filtertid*)
	_LG_FL					:INT;		(* Larmfördröjning givarfel *)
END_VAR

VAR_OUTPUT
	_rMV						:REAL;		(* Mätvärde *)
	_bLG						:BOOL; 	(*Givarfel*)
	_bDelayedLG				:BOOL;	(* Fördröjt givarfel *)
END_VAR
(* body not read: cfc101 *)
END_PROGRAM

(* POU _IOs_Uppdelat_per_skåp/HUS1_AS02/_IO/ANALOGA IN/Kort04/HUS1_AS02_Analoga_in_Kort04_AI04, FAI *)
PROGRAM HUS1_AS02_Analoga_in_Kort04_AI04
(*#####################################   Temperature Sensor Ex2   ################################################################*)
VAR
	(*===========================Configuration of terminal==========================================*)
	fbConfigureKL32xx					:FB_HVACConfigureKL32xx;
	_byCtrlKL32xx                         			AT %Q*: BYTE;
	_iDataOutKL32xx                       		AT %Q*: INT;
	_iDataInKL32xx 					AT%I*:INT;(* Raw Value from the Terminal *)
	_byStatusKL32xx 			AT%I*:BYTE;(* Statusbyte from Terminal *)

	_bScanSensor              					: BOOL;
	_tTimeOut                 					: TIME := T#5s;
	_bSetSensor               					: BOOL;
	bReady                               				: BOOL;
	byOutStatus                          			: BYTE;
	iOutDataIn                           				: INT;
	_eBusTerminalKL32xx                   		: E_HVACBusTerminal_KL32xx;
	_eStatusScanSensorType                	: E_HVACSensorType;
	_bErrorGeneral                        			: BOOL;
	_byError                              				: BYTE;
	_bErrorCommunication                  		: BOOL;
	_bErrorBusTerminalNotSupported   	: BOOL;
	_bErrorSensorType                     		: BOOL;
	_bErrorScanSensor                     		: BOOL;
	(*========================================================================================*)

	_bReset_Local					:BOOL;
	_bSetDefaultTempSens			:BOOL;

	(*========================================================================================*)
	FBHVACTemperatureSensor: FB_HVACTemperatureSensor;
	eDataSecurityType					: E_HVACDataSecurityType:=1;
	bSetDefault								:BOOL;
	iRawValue								:INT;
	byStatusRawValue						:BYTE;
	bEnableLimitCtrl							:BOOL;
	bReset									:BOOL;
	bErrorGeneral					:BOOL;
	byError							:BYTE;
	bErrorShortCircuit				:BOOL;
	bErrorBrokenSensor				:BOOL;
	bErrorHighLimit					:BOOL;
	bErrorLowLimit					:BOOL;
	bErrorCycleTime					:BOOL;
	bInvalidParameter				:BOOL;
	rOffset									:REAL;
	rHighLimit								:REAL;
	rLowLimit								:REAL;
	rReplacementValue						:REAL;
	tFilterTime								:TIME;
	eTemperatureSensorMode				:E_HVACTemperatureSensorMode:=2;
	fbAlarmD: fbDelayedAlarmMinutes;

END_VAR

VAR_INPUT
	_rKAL						: REAL;	(*Kalibrering*)
	_FT						:INT;		(*Filtertid*)
	_LG_FL					:INT;		(* Larmfördröjning givarfel *)
END_VAR

VAR_OUTPUT
	_rMV						:REAL;		(* Mätvärde *)
	_bLG						:BOOL; 	(*Givarfel*)
	_bDelayedLG				:BOOL;	(* Fördröjt givarfel *)
END_VAR
(* body not read: cfc101 *)
END_PROGRAM

(* POU _IOs_Uppdelat_per_skåp/HUS1_AS02/_IO/ANALOGA IN/Kort04/HUS1_AS02_Analoga_in_Kort04_AI08, FAI *)
PROGRAM HUS1_AS02_Analoga_in_Kort04_AI08
(*#####################################   Temperature Sensor Ex2   ################################################################*)
VAR
	(*===========================Configuration of terminal==========================================*)
	fbConfigureKL32xx					:FB_HVACConfigureKL32xx;
	_byCtrlKL32xx                         			AT %Q*: BYTE;
	_iDataOutKL32xx                       		AT %Q*: INT;
	_iDataInKL32xx 					AT%I*:INT;(* Raw Value from the Terminal *)
	_byStatusKL32xx 			AT%I*:BYTE;(* Statusbyte from Terminal *)

	_bScanSensor              					: BOOL;
	_tTimeOut                 					: TIME := T#5s;
	_bSetSensor               					: BOOL;
	bReady                               				: BOOL;
	byOutStatus                          			: BYTE;
	iOutDataIn                           				: INT;
	_eBusTerminalKL32xx                   		: E_HVACBusTerminal_KL32xx;
	_eStatusScanSensorType                	: E_HVACSensorType;
	_bErrorGeneral                        			: BOOL;
	_byError                              				: BYTE;
	_bErrorCommunication                  		: BOOL;
	_bErrorBusTerminalNotSupported   	: BOOL;
	_bErrorSensorType                     		: BOOL;
	_bErrorScanSensor                     		: BOOL;
	(*========================================================================================*)

	_bReset_Local					:BOOL;
	_bSetDefaultTempSens			:BOOL;

	(*========================================================================================*)
	FBHVACTemperatureSensor: FB_HVACTemperatureSensor;
	eDataSecurityType					: E_HVACDataSecurityType:=1;
	bSetDefault								:BOOL;
	iRawValue								:INT;
	byStatusRawValue						:BYTE;
	bEnableLimitCtrl							:BOOL;
	bReset									:BOOL;
	bErrorGeneral					:BOOL;
	byError							:BYTE;
	bErrorShortCircuit				:BOOL;
	bErrorBrokenSensor				:BOOL;
	bErrorHighLimit					:BOOL;
	bErrorLowLimit					:BOOL;
	bErrorCycleTime					:BOOL;
	bInvalidParameter				:BOOL;
	rOffset									:REAL;
	rHighLimit								:REAL;
	rLowLimit								:REAL;
	rReplacementValue						:REAL;
	tFilterTime								:TIME;
	eTemperatureSensorMode				:E_HVACTemperatureSensorMode:=2;
	fbAlarmD: fbDelayedAlarmMinutes;

END_VAR

VAR_INPUT
	_rKAL						: REAL;	(*Kalibrering*)
	_FT						:INT;		(*Filtertid*)
	_LG_FL					:INT;		(* Larmfördröjning givarfel *)
END_VAR

VAR_OUTPUT
	_rMV						:REAL;		(* Mätvärde *)
	_bLG						:BOOL; 	(*Givarfel*)
	_bDelayedLG				:BOOL;	(* Fördröjt givarfel *)
END_VAR
(* body not read: cfc101 *)
END_PROGRAM

(* POU _IOs_Uppdelat_per_skåp/HUS1_AS02/_IO/ANALOGA UT/Kort05/HUS1_AS02_Analoga_ut_Kort05, CFC *)
PROGRAM HUS1_AS02_Analoga_ut_Kort05
VAR

	Conversion_AU1: fbConversionScale;
	Conversion_AU2: fbConversionScale;
	Conversion_AU3: fbConversionScale;
	Conversion_AU4: fbConversionScale;
	Conversion_AU5: fbConversionScale;
	Conversion_AU6: fbConversionScale;
	Conversion_AU7: fbConversionScale;
	Conversion_AU8: fbConversionScale;

END_VAR
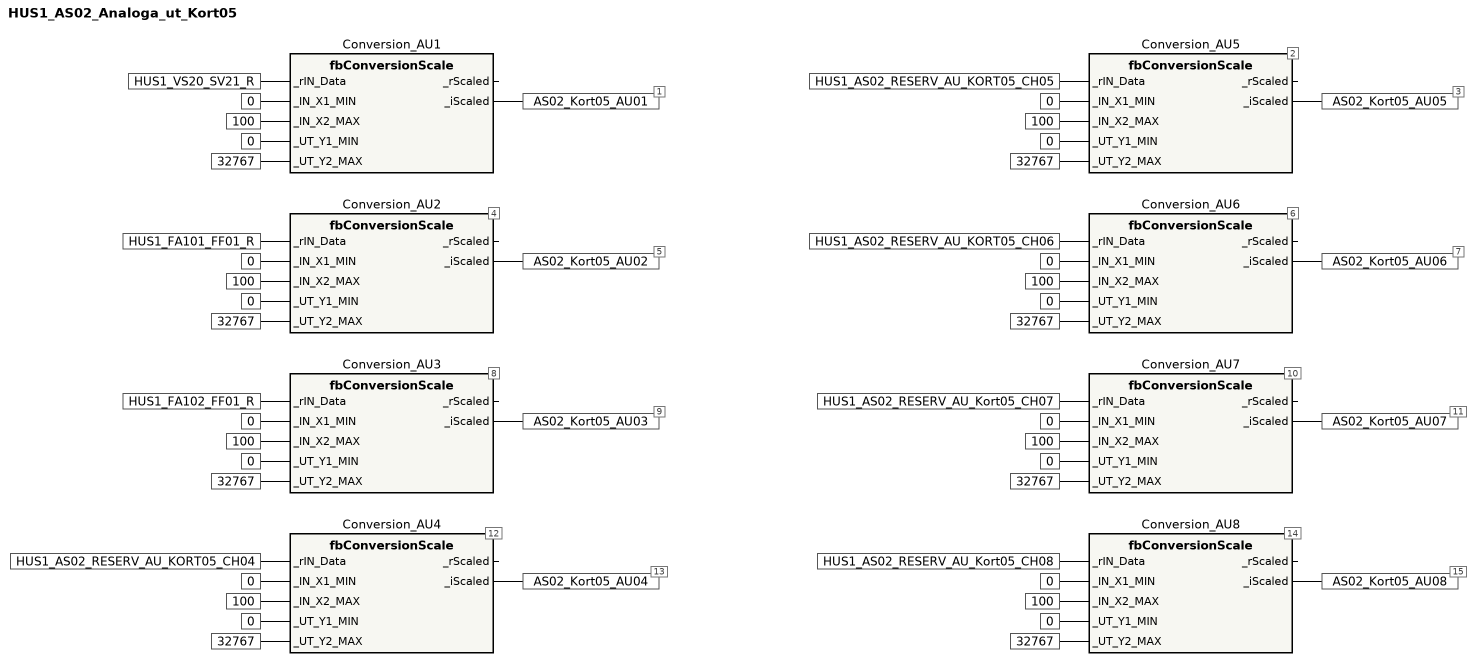
_CFC_ (* Continuous Function Chart, elements in execution order *)
#0 Conversion_AU1:fbConversionScale(_rIN_Data: HUS1_VS20_SV21_R, _IN_X1_MIN: 0, _IN_X2_MAX: 100, _UT_Y1_MIN: 0, _UT_Y2_MAX: 32767)
#1 AS02_Kort05_AU01 <= #0._iScaled
#2 Conversion_AU5:fbConversionScale(_rIN_Data: HUS1_AS02_RESERV_AU_KORT05_CH05, _IN_X1_MIN: 0, _IN_X2_MAX: 100, _UT_Y1_MIN: 0, _UT_Y2_MAX: 32767)
#3 AS02_Kort05_AU05 <= #2._iScaled
#4 Conversion_AU2:fbConversionScale(_rIN_Data: HUS1_FA101_FF01_R, _IN_X1_MIN: 0, _IN_X2_MAX: 100, _UT_Y1_MIN: 0, _UT_Y2_MAX: 32767)
#5 AS02_Kort05_AU02 <= #4._iScaled
#6 Conversion_AU6:fbConversionScale(_rIN_Data: HUS1_AS02_RESERV_AU_KORT05_CH06, _IN_X1_MIN: 0, _IN_X2_MAX: 100, _UT_Y1_MIN: 0, _UT_Y2_MAX: 32767)
#7 AS02_Kort05_AU06 <= #6._iScaled
#8 Conversion_AU3:fbConversionScale(_rIN_Data: HUS1_FA102_FF01_R, _IN_X1_MIN: 0, _IN_X2_MAX: 100, _UT_Y1_MIN: 0, _UT_Y2_MAX: 32767)
#9 AS02_Kort05_AU03 <= #8._iScaled
#10 Conversion_AU7:fbConversionScale(_rIN_Data: HUS1_AS02_RESERV_AU_Kort05_CH07, _IN_X1_MIN: 0, _IN_X2_MAX: 100, _UT_Y1_MIN: 0, _UT_Y2_MAX: 32767)
#11 AS02_Kort05_AU07 <= #10._iScaled
#12 Conversion_AU4:fbConversionScale(_rIN_Data: HUS1_AS02_RESERV_AU_KORT05_CH04, _IN_X1_MIN: 0, _IN_X2_MAX: 100, _UT_Y1_MIN: 0, _UT_Y2_MAX: 32767)
#13 AS02_Kort05_AU04 <= #12._iScaled
#14 Conversion_AU8:fbConversionScale(_rIN_Data: HUS1_AS02_RESERV_AU_Kort05_CH08, _IN_X1_MIN: 0, _IN_X2_MAX: 100, _UT_Y1_MIN: 0, _UT_Y2_MAX: 32767)
#15 AS02_Kort05_AU08 <= #14._iScaled
_END_CFC_
(* the same logic as Structured Text *)
Conversion_AU1(_rIN_Data := HUS1_VS20_SV21_R, _IN_X1_MIN := 0, _IN_X2_MAX := 100, _UT_Y1_MIN := 0, _UT_Y2_MAX := 32767);
AS02_Kort05_AU01 := Conversion_AU1._iScaled;
Conversion_AU5(_rIN_Data := HUS1_AS02_RESERV_AU_KORT05_CH05, _IN_X1_MIN := 0, _IN_X2_MAX := 100, _UT_Y1_MIN := 0, _UT_Y2_MAX := 32767);
AS02_Kort05_AU05 := Conversion_AU5._iScaled;
Conversion_AU2(_rIN_Data := HUS1_FA101_FF01_R, _IN_X1_MIN := 0, _IN_X2_MAX := 100, _UT_Y1_MIN := 0, _UT_Y2_MAX := 32767);
AS02_Kort05_AU02 := Conversion_AU2._iScaled;
Conversion_AU6(_rIN_Data := HUS1_AS02_RESERV_AU_KORT05_CH06, _IN_X1_MIN := 0, _IN_X2_MAX := 100, _UT_Y1_MIN := 0, _UT_Y2_MAX := 32767);
AS02_Kort05_AU06 := Conversion_AU6._iScaled;
Conversion_AU3(_rIN_Data := HUS1_FA102_FF01_R, _IN_X1_MIN := 0, _IN_X2_MAX := 100, _UT_Y1_MIN := 0, _UT_Y2_MAX := 32767);
AS02_Kort05_AU03 := Conversion_AU3._iScaled;
Conversion_AU7(_rIN_Data := HUS1_AS02_RESERV_AU_Kort05_CH07, _IN_X1_MIN := 0, _IN_X2_MAX := 100, _UT_Y1_MIN := 0, _UT_Y2_MAX := 32767);
AS02_Kort05_AU07 := Conversion_AU7._iScaled;
Conversion_AU4(_rIN_Data := HUS1_AS02_RESERV_AU_KORT05_CH04, _IN_X1_MIN := 0, _IN_X2_MAX := 100, _UT_Y1_MIN := 0, _UT_Y2_MAX := 32767);
AS02_Kort05_AU04 := Conversion_AU4._iScaled;
Conversion_AU8(_rIN_Data := HUS1_AS02_RESERV_AU_Kort05_CH08, _IN_X1_MIN := 0, _IN_X2_MAX := 100, _UT_Y1_MIN := 0, _UT_Y2_MAX := 32767);
AS02_Kort05_AU08 := Conversion_AU8._iScaled;
END_PROGRAM

(* POU xEgna Funktionsblock/fbConversionScale, CFC *)
FUNCTION_BLOCK fbConversionScale
VAR
	fbSkalaUtsignal: FB_HVACScale;
	Default						:BOOL;

END_VAR

VAR_INPUT
	_rIN_Data					:REAL;
	_IN_X1_MIN				:REAL;
	_IN_X2_MAX			:REAL;
	_UT_Y1_MIN				:REAL;
	_UT_Y2_MAX			:REAL;
END_VAR

VAR_OUTPUT
	_rScaled					:REAL;
	_iScaled					:INT;
END_VAR
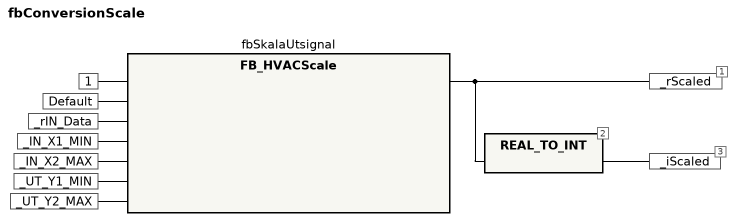
_CFC_ (* Continuous Function Chart, elements in execution order *)
#0 fbSkalaUtsignal:FB_HVACScale(1, Default, _rIN_Data, _IN_X1_MIN, _IN_X2_MAX, _UT_Y1_MIN, _UT_Y2_MAX)
#1 _rScaled <= #0
#2 REAL_TO_INT(#0)
#3 _iScaled <= #2
_END_CFC_
END_FUNCTION_BLOCK

(* POU _IOs_Uppdelat_per_skåp/HUS2_AS01/_IO/HUS2_AS01_IO_MAIN, CFC *)
PROGRAM HUS2_AS01_IO_MAIN
VAR
END_VAR
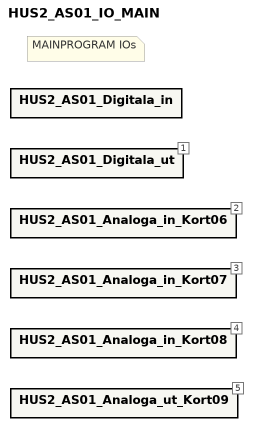
_CFC_ (* Continuous Function Chart, elements in execution order *)
(* MAINPROGRAM IOs *)
#0 HUS2_AS01_Digitala_in()
#1 HUS2_AS01_Digitala_ut()
#2 HUS2_AS01_Analoga_in_Kort06()
#3 HUS2_AS01_Analoga_in_Kort07()
#4 HUS2_AS01_Analoga_in_Kort08()
#5 HUS2_AS01_Analoga_ut_Kort09()
_END_CFC_
(* the same logic as Structured Text *)
(* MAINPROGRAM IOs *)
HUS2_AS01_Digitala_in();
HUS2_AS01_Digitala_ut();
HUS2_AS01_Analoga_in_Kort06();
HUS2_AS01_Analoga_in_Kort07();
HUS2_AS01_Analoga_in_Kort08();
HUS2_AS01_Analoga_ut_Kort09();
END_PROGRAM

(* POU _IOs_Uppdelat_per_skåp/HUS2_AS01/_IO/HUS2_AS01_Digitala_in, CFC *)
PROGRAM HUS2_AS01_Digitala_in

VAR


END_VAR
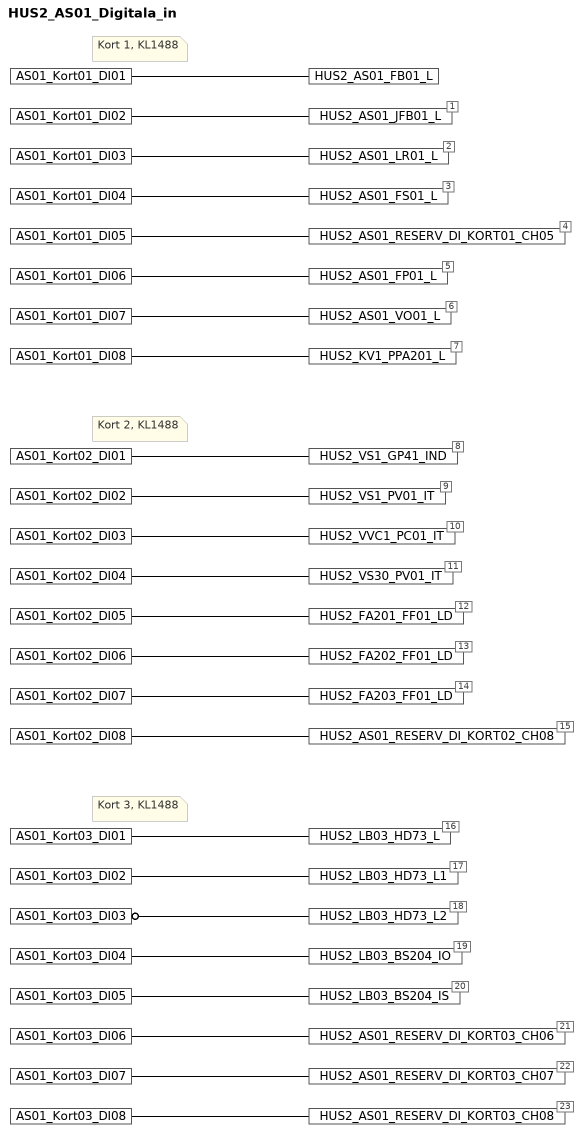
_CFC_ (* Continuous Function Chart, elements in execution order *)
(* Kort 3, KL1488 *)
(* Kort 1, KL1488 *)
(* Kort 2, KL1488 *)
#0 HUS2_AS01_FB01_L <= AS01_Kort01_DI01
#1 HUS2_AS01_JFB01_L <= AS01_Kort01_DI02
#2 HUS2_AS01_LR01_L <= AS01_Kort01_DI03
#3 HUS2_AS01_FS01_L <= AS01_Kort01_DI04
#4 HUS2_AS01_RESERV_DI_KORT01_CH05 <= AS01_Kort01_DI05
#5 HUS2_AS01_FP01_L <= AS01_Kort01_DI06
#6 HUS2_AS01_VO01_L <= AS01_Kort01_DI07
#7 HUS2_KV1_PPA201_L <= AS01_Kort01_DI08
#8 HUS2_VS1_GP41_IND <= AS01_Kort02_DI01
#9 HUS2_VS1_PV01_IT <= AS01_Kort02_DI02
#10 HUS2_VVC1_PC01_IT <= AS01_Kort02_DI03
#11 HUS2_VS30_PV01_IT <= AS01_Kort02_DI04
#12 HUS2_FA201_FF01_LD <= AS01_Kort02_DI05
#13 HUS2_FA202_FF01_LD <= AS01_Kort02_DI06
#14 HUS2_FA203_FF01_LD <= AS01_Kort02_DI07
#15 HUS2_AS01_RESERV_DI_KORT02_CH08 <= AS01_Kort02_DI08
#16 HUS2_LB03_HD73_L <= AS01_Kort03_DI01
#17 HUS2_LB03_HD73_L1 <= AS01_Kort03_DI02
#18 HUS2_LB03_HD73_L2 <= NOT AS01_Kort03_DI03
#19 HUS2_LB03_BS204_IO <= AS01_Kort03_DI04
#20 HUS2_LB03_BS204_IS <= AS01_Kort03_DI05
#21 HUS2_AS01_RESERV_DI_KORT03_CH06 <= AS01_Kort03_DI06
#22 HUS2_AS01_RESERV_DI_KORT03_CH07 <= AS01_Kort03_DI07
#23 HUS2_AS01_RESERV_DI_KORT03_CH08 <= AS01_Kort03_DI08
_END_CFC_
(* the same logic as Structured Text *)
(* Kort 3, KL1488 *)
(* Kort 1, KL1488 *)
(* Kort 2, KL1488 *)
HUS2_AS01_FB01_L := AS01_Kort01_DI01;
HUS2_AS01_JFB01_L := AS01_Kort01_DI02;
HUS2_AS01_LR01_L := AS01_Kort01_DI03;
HUS2_AS01_FS01_L := AS01_Kort01_DI04;
HUS2_AS01_RESERV_DI_KORT01_CH05 := AS01_Kort01_DI05;
HUS2_AS01_FP01_L := AS01_Kort01_DI06;
HUS2_AS01_VO01_L := AS01_Kort01_DI07;
HUS2_KV1_PPA201_L := AS01_Kort01_DI08;
HUS2_VS1_GP41_IND := AS01_Kort02_DI01;
HUS2_VS1_PV01_IT := AS01_Kort02_DI02;
HUS2_VVC1_PC01_IT := AS01_Kort02_DI03;
HUS2_VS30_PV01_IT := AS01_Kort02_DI04;
HUS2_FA201_FF01_LD := AS01_Kort02_DI05;
HUS2_FA202_FF01_LD := AS01_Kort02_DI06;
HUS2_FA203_FF01_LD := AS01_Kort02_DI07;
HUS2_AS01_RESERV_DI_KORT02_CH08 := AS01_Kort02_DI08;
HUS2_LB03_HD73_L := AS01_Kort03_DI01;
HUS2_LB03_HD73_L1 := AS01_Kort03_DI02;
HUS2_LB03_HD73_L2 := NOT AS01_Kort03_DI03;
HUS2_LB03_BS204_IO := AS01_Kort03_DI04;
HUS2_LB03_BS204_IS := AS01_Kort03_DI05;
HUS2_AS01_RESERV_DI_KORT03_CH06 := AS01_Kort03_DI06;
HUS2_AS01_RESERV_DI_KORT03_CH07 := AS01_Kort03_DI07;
HUS2_AS01_RESERV_DI_KORT03_CH08 := AS01_Kort03_DI08;
END_PROGRAM

(* POU _IOs_Uppdelat_per_skåp/HUS2_AS01/_IO/HUS2_AS01_Digitala_ut, CFC *)
PROGRAM HUS2_AS01_Digitala_ut


VAR
END_VAR
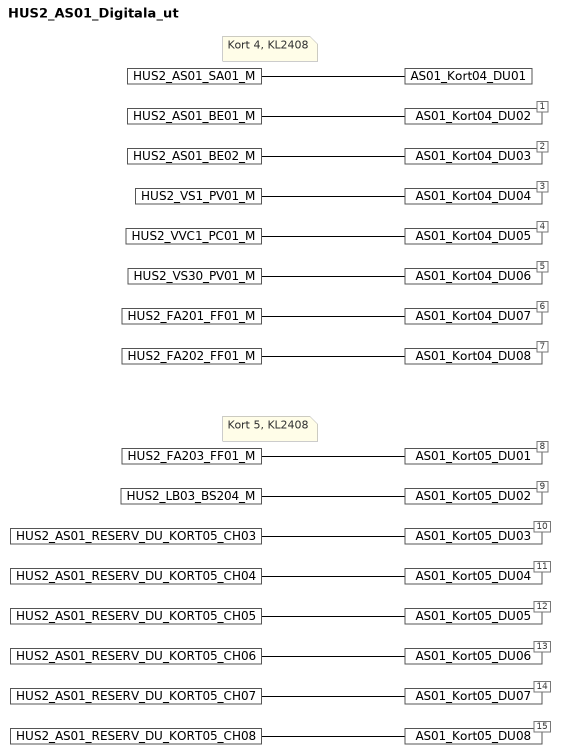
_CFC_ (* Continuous Function Chart, elements in execution order *)
(* Kort 4, KL2408 *)
(* Kort 5, KL2408 *)
#0 AS01_Kort04_DU01 <= HUS2_AS01_SA01_M
#1 AS01_Kort04_DU02 <= HUS2_AS01_BE01_M
#2 AS01_Kort04_DU03 <= HUS2_AS01_BE02_M
#3 AS01_Kort04_DU04 <= HUS2_VS1_PV01_M
#4 AS01_Kort04_DU05 <= HUS2_VVC1_PC01_M
#5 AS01_Kort04_DU06 <= HUS2_VS30_PV01_M
#6 AS01_Kort04_DU07 <= HUS2_FA201_FF01_M
#7 AS01_Kort04_DU08 <= HUS2_FA202_FF01_M
#8 AS01_Kort05_DU01 <= HUS2_FA203_FF01_M
#9 AS01_Kort05_DU02 <= HUS2_LB03_BS204_M
#10 AS01_Kort05_DU03 <= HUS2_AS01_RESERV_DU_KORT05_CH03
#11 AS01_Kort05_DU04 <= HUS2_AS01_RESERV_DU_KORT05_CH04
#12 AS01_Kort05_DU05 <= HUS2_AS01_RESERV_DU_KORT05_CH05
#13 AS01_Kort05_DU06 <= HUS2_AS01_RESERV_DU_KORT05_CH06
#14 AS01_Kort05_DU07 <= HUS2_AS01_RESERV_DU_KORT05_CH07
#15 AS01_Kort05_DU08 <= HUS2_AS01_RESERV_DU_KORT05_CH08
_END_CFC_
(* the same logic as Structured Text *)
(* Kort 4, KL2408 *)
(* Kort 5, KL2408 *)
AS01_Kort04_DU01 := HUS2_AS01_SA01_M;
AS01_Kort04_DU02 := HUS2_AS01_BE01_M;
AS01_Kort04_DU03 := HUS2_AS01_BE02_M;
AS01_Kort04_DU04 := HUS2_VS1_PV01_M;
AS01_Kort04_DU05 := HUS2_VVC1_PC01_M;
AS01_Kort04_DU06 := HUS2_VS30_PV01_M;
AS01_Kort04_DU07 := HUS2_FA201_FF01_M;
AS01_Kort04_DU08 := HUS2_FA202_FF01_M;
AS01_Kort05_DU01 := HUS2_FA203_FF01_M;
AS01_Kort05_DU02 := HUS2_LB03_BS204_M;
AS01_Kort05_DU03 := HUS2_AS01_RESERV_DU_KORT05_CH03;
AS01_Kort05_DU04 := HUS2_AS01_RESERV_DU_KORT05_CH04;
AS01_Kort05_DU05 := HUS2_AS01_RESERV_DU_KORT05_CH05;
AS01_Kort05_DU06 := HUS2_AS01_RESERV_DU_KORT05_CH06;
AS01_Kort05_DU07 := HUS2_AS01_RESERV_DU_KORT05_CH07;
AS01_Kort05_DU08 := HUS2_AS01_RESERV_DU_KORT05_CH08;
END_PROGRAM

(* POU _IOs_Uppdelat_per_skåp/HUS2_AS01/_IO/ANALOGA IN/Kort06/HUS2_AS01_Analoga_in_Kort06, CFC *)
PROGRAM HUS2_AS01_Analoga_in_Kort06
VAR
	bLG01: BOOL;
	bLG02: BOOL;
	bLG03: BOOL;
	bLG04: BOOL;
	bLG05: BOOL;
	bLG06: BOOL;
	bLG07: BOOL;
	bLG08: BOOL;

(*TEMP*)
	FT1:INT;
	LG_FL1:INT;
	FT2:INT;
	LG_FL2:INT;
	FT3:INT;
	LG_FL3:INT;
	FT4:INT;
	LG_FL4:INT;
	FT5:INT;
	LG_FL5:INT;
	FT6:INT;
	LG_FL6:INT;
	FT7:INT;
	LG_FL7:INT;
	FT8:INT;
	LG_FL8:INT;

END_VAR
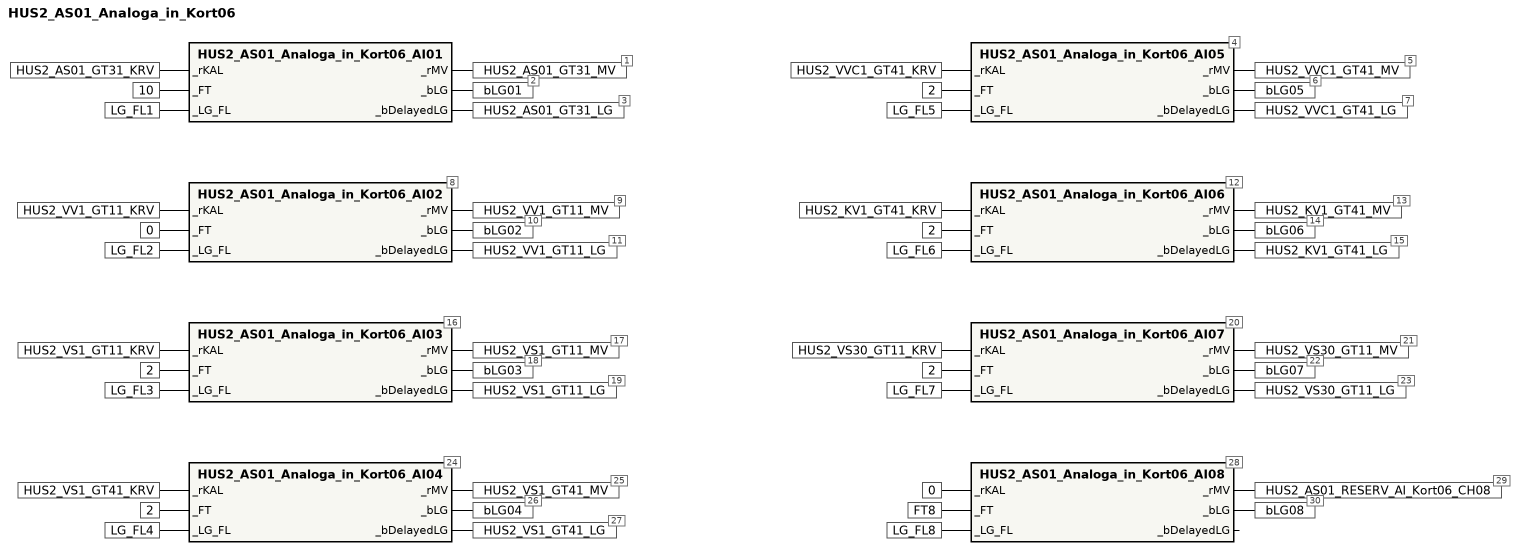
_CFC_ (* Continuous Function Chart, elements in execution order *)
#0 HUS2_AS01_Analoga_in_Kort06_AI01(_rKAL: HUS2_AS01_GT31_KRV, _FT: 10, _LG_FL: LG_FL1)
#1 HUS2_AS01_GT31_MV <= #0._rMV
#2 bLG01 <= #0._bLG
#3 HUS2_AS01_GT31_LG <= #0._bDelayedLG
#4 HUS2_AS01_Analoga_in_Kort06_AI05(_rKAL: HUS2_VVC1_GT41_KRV, _FT: 2, _LG_FL: LG_FL5)
#5 HUS2_VVC1_GT41_MV <= #4._rMV
#6 bLG05 <= #4._bLG
#7 HUS2_VVC1_GT41_LG <= #4._bDelayedLG
#8 HUS2_AS01_Analoga_in_Kort06_AI02(_rKAL: HUS2_VV1_GT11_KRV, _FT: 0, _LG_FL: LG_FL2)
#9 HUS2_VV1_GT11_MV <= #8._rMV
#10 bLG02 <= #8._bLG
#11 HUS2_VV1_GT11_LG <= #8._bDelayedLG
#12 HUS2_AS01_Analoga_in_Kort06_AI06(_rKAL: HUS2_KV1_GT41_KRV, _FT: 2, _LG_FL: LG_FL6)
#13 HUS2_KV1_GT41_MV <= #12._rMV
#14 bLG06 <= #12._bLG
#15 HUS2_KV1_GT41_LG <= #12._bDelayedLG
#16 HUS2_AS01_Analoga_in_Kort06_AI03(_rKAL: HUS2_VS1_GT11_KRV, _FT: 2, _LG_FL: LG_FL3)
#17 HUS2_VS1_GT11_MV <= #16._rMV
#18 bLG03 <= #16._bLG
#19 HUS2_VS1_GT11_LG <= #16._bDelayedLG
#20 HUS2_AS01_Analoga_in_Kort06_AI07(_rKAL: HUS2_VS30_GT11_KRV, _FT: 2, _LG_FL: LG_FL7)
#21 HUS2_VS30_GT11_MV <= #20._rMV
#22 bLG07 <= #20._bLG
#23 HUS2_VS30_GT11_LG <= #20._bDelayedLG
#24 HUS2_AS01_Analoga_in_Kort06_AI04(_rKAL: HUS2_VS1_GT41_KRV, _FT: 2, _LG_FL: LG_FL4)
#25 HUS2_VS1_GT41_MV <= #24._rMV
#26 bLG04 <= #24._bLG
#27 HUS2_VS1_GT41_LG <= #24._bDelayedLG
#28 HUS2_AS01_Analoga_in_Kort06_AI08(_rKAL: 0, _FT: FT8, _LG_FL: LG_FL8)
#29 HUS2_AS01_RESERV_AI_Kort06_CH08 <= #28._rMV
#30 bLG08 <= #28._bLG
_END_CFC_
(* the same logic as Structured Text *)
HUS2_AS01_Analoga_in_Kort06_AI01(_rKAL := HUS2_AS01_GT31_KRV, _FT := 10, _LG_FL := LG_FL1);
HUS2_AS01_GT31_MV := HUS2_AS01_Analoga_in_Kort06_AI01._rMV;
bLG01 := HUS2_AS01_Analoga_in_Kort06_AI01._bLG;
HUS2_AS01_GT31_LG := HUS2_AS01_Analoga_in_Kort06_AI01._bDelayedLG;
HUS2_AS01_Analoga_in_Kort06_AI05(_rKAL := HUS2_VVC1_GT41_KRV, _FT := 2, _LG_FL := LG_FL5);
HUS2_VVC1_GT41_MV := HUS2_AS01_Analoga_in_Kort06_AI05._rMV;
bLG05 := HUS2_AS01_Analoga_in_Kort06_AI05._bLG;
HUS2_VVC1_GT41_LG := HUS2_AS01_Analoga_in_Kort06_AI05._bDelayedLG;
HUS2_AS01_Analoga_in_Kort06_AI02(_rKAL := HUS2_VV1_GT11_KRV, _FT := 0, _LG_FL := LG_FL2);
HUS2_VV1_GT11_MV := HUS2_AS01_Analoga_in_Kort06_AI02._rMV;
bLG02 := HUS2_AS01_Analoga_in_Kort06_AI02._bLG;
HUS2_VV1_GT11_LG := HUS2_AS01_Analoga_in_Kort06_AI02._bDelayedLG;
HUS2_AS01_Analoga_in_Kort06_AI06(_rKAL := HUS2_KV1_GT41_KRV, _FT := 2, _LG_FL := LG_FL6);
HUS2_KV1_GT41_MV := HUS2_AS01_Analoga_in_Kort06_AI06._rMV;
bLG06 := HUS2_AS01_Analoga_in_Kort06_AI06._bLG;
HUS2_KV1_GT41_LG := HUS2_AS01_Analoga_in_Kort06_AI06._bDelayedLG;
HUS2_AS01_Analoga_in_Kort06_AI03(_rKAL := HUS2_VS1_GT11_KRV, _FT := 2, _LG_FL := LG_FL3);
HUS2_VS1_GT11_MV := HUS2_AS01_Analoga_in_Kort06_AI03._rMV;
bLG03 := HUS2_AS01_Analoga_in_Kort06_AI03._bLG;
HUS2_VS1_GT11_LG := HUS2_AS01_Analoga_in_Kort06_AI03._bDelayedLG;
HUS2_AS01_Analoga_in_Kort06_AI07(_rKAL := HUS2_VS30_GT11_KRV, _FT := 2, _LG_FL := LG_FL7);
HUS2_VS30_GT11_MV := HUS2_AS01_Analoga_in_Kort06_AI07._rMV;
bLG07 := HUS2_AS01_Analoga_in_Kort06_AI07._bLG;
HUS2_VS30_GT11_LG := HUS2_AS01_Analoga_in_Kort06_AI07._bDelayedLG;
HUS2_AS01_Analoga_in_Kort06_AI04(_rKAL := HUS2_VS1_GT41_KRV, _FT := 2, _LG_FL := LG_FL4);
HUS2_VS1_GT41_MV := HUS2_AS01_Analoga_in_Kort06_AI04._rMV;
bLG04 := HUS2_AS01_Analoga_in_Kort06_AI04._bLG;
HUS2_VS1_GT41_LG := HUS2_AS01_Analoga_in_Kort06_AI04._bDelayedLG;
HUS2_AS01_Analoga_in_Kort06_AI08(_rKAL := 0, _FT := FT8, _LG_FL := LG_FL8);
HUS2_AS01_RESERV_AI_Kort06_CH08 := HUS2_AS01_Analoga_in_Kort06_AI08._rMV;
bLG08 := HUS2_AS01_Analoga_in_Kort06_AI08._bLG;
END_PROGRAM

(* POU _IOs_Uppdelat_per_skåp/HUS2_AS01/_IO/ANALOGA IN/Kort06/HUS2_AS01_Analoga_in_Kort06_AI01, FAI *)
PROGRAM HUS2_AS01_Analoga_in_Kort06_AI01
(*#####################################   Temperature Sensor Ex2   ################################################################*)
VAR
	(*===========================Configuration of terminal==========================================*)
	fbConfigureKL32xx					:FB_HVACConfigureKL32xx;
	_byCtrlKL32xx                         			AT %Q*: BYTE;
	_iDataOutKL32xx                       		AT %Q*: INT;
	_iDataInKL32xx 					AT%I*:INT;(* Raw Value from the Terminal *)
	_byStatusKL32xx 			AT%I*:BYTE;(* Statusbyte from Terminal *)

	_bScanSensor              					: BOOL;
	_tTimeOut                 					: TIME := T#5s;
	_bSetSensor               					: BOOL;
	bReady                               				: BOOL;
	byOutStatus                          			: BYTE;
	iOutDataIn                           				: INT;
	_eBusTerminalKL32xx                   		: E_HVACBusTerminal_KL32xx;
	_eStatusScanSensorType                	: E_HVACSensorType;
	_bErrorGeneral                        			: BOOL;
	_byError                              				: BYTE;
	_bErrorCommunication                  		: BOOL;
	_bErrorBusTerminalNotSupported   	: BOOL;
	_bErrorSensorType                     		: BOOL;
	_bErrorScanSensor                     		: BOOL;
	(*========================================================================================*)

	_bReset_Local					:BOOL;
	_bSetDefaultTempSens			:BOOL;

	(*========================================================================================*)
	FBHVACTemperatureSensor: FB_HVACTemperatureSensor;
	eDataSecurityType					: E_HVACDataSecurityType:=1;
	bSetDefault								:BOOL;
	iRawValue								:INT;
	byStatusRawValue						:BYTE;
	bEnableLimitCtrl							:BOOL;
	bReset									:BOOL;
	bErrorGeneral					:BOOL;
	byError							:BYTE;
	bErrorShortCircuit				:BOOL;
	bErrorBrokenSensor				:BOOL;
	bErrorHighLimit					:BOOL;
	bErrorLowLimit					:BOOL;
	bErrorCycleTime					:BOOL;
	bInvalidParameter				:BOOL;
	rOffset									:REAL;
	rHighLimit								:REAL;
	rLowLimit								:REAL;
	rReplacementValue						:REAL;
	tFilterTime								:TIME;
	eTemperatureSensorMode				:E_HVACTemperatureSensorMode:=2;
	fbAlarmD: fbDelayedAlarmMinutes;

END_VAR

VAR_INPUT
	_rKAL						: REAL;	(*Kalibrering*)
	_FT						:INT;		(*Filtertid*)
	_LG_FL					:INT;		(* Larmfördröjning givarfel *)
END_VAR

VAR_OUTPUT
	_rMV						:REAL;		(* Mätvärde *)
	_bLG						:BOOL; 	(*Givarfel*)
	_bDelayedLG				:BOOL;	(* Fördröjt givarfel *)
END_VAR
(* body not read: cfc101 *)
END_PROGRAM

(* POU _IOs_Uppdelat_per_skåp/HUS2_AS01/_IO/ANALOGA IN/Kort06/HUS2_AS01_Analoga_in_Kort06_AI05, FAI *)
PROGRAM HUS2_AS01_Analoga_in_Kort06_AI05
(*#####################################   Temperature Sensor Ex2   ################################################################*)
VAR
	(*===========================Configuration of terminal==========================================*)
	fbConfigureKL32xx					:FB_HVACConfigureKL32xx;
	_byCtrlKL32xx                         			AT %Q*: BYTE;
	_iDataOutKL32xx                       		AT %Q*: INT;
	_iDataInKL32xx 					AT%I*:INT;(* Raw Value from the Terminal *)
	_byStatusKL32xx 			AT%I*:BYTE;(* Statusbyte from Terminal *)

	_bScanSensor              					: BOOL;
	_tTimeOut                 					: TIME := T#5s;
	_bSetSensor               					: BOOL;
	bReady                               				: BOOL;
	byOutStatus                          			: BYTE;
	iOutDataIn                           				: INT;
	_eBusTerminalKL32xx                   		: E_HVACBusTerminal_KL32xx;
	_eStatusScanSensorType                	: E_HVACSensorType;
	_bErrorGeneral                        			: BOOL;
	_byError                              				: BYTE;
	_bErrorCommunication                  		: BOOL;
	_bErrorBusTerminalNotSupported   	: BOOL;
	_bErrorSensorType                     		: BOOL;
	_bErrorScanSensor                     		: BOOL;
	(*========================================================================================*)

	_bReset_Local					:BOOL;
	_bSetDefaultTempSens			:BOOL;

	(*========================================================================================*)
	FBHVACTemperatureSensor: FB_HVACTemperatureSensor;
	eDataSecurityType					: E_HVACDataSecurityType:=1;
	bSetDefault								:BOOL;
	iRawValue								:INT;
	byStatusRawValue						:BYTE;
	bEnableLimitCtrl							:BOOL;
	bReset									:BOOL;
	bErrorGeneral					:BOOL;
	byError							:BYTE;
	bErrorShortCircuit				:BOOL;
	bErrorBrokenSensor				:BOOL;
	bErrorHighLimit					:BOOL;
	bErrorLowLimit					:BOOL;
	bErrorCycleTime					:BOOL;
	bInvalidParameter				:BOOL;
	rOffset									:REAL;
	rHighLimit								:REAL;
	rLowLimit								:REAL;
	rReplacementValue						:REAL;
	tFilterTime								:TIME;
	eTemperatureSensorMode				:E_HVACTemperatureSensorMode:=2;
	fbAlarmD: fbDelayedAlarmMinutes;

END_VAR

VAR_INPUT
	_rKAL						: REAL;	(*Kalibrering*)
	_FT						:INT;		(*Filtertid*)
	_LG_FL					:INT;		(* Larmfördröjning givarfel *)
END_VAR

VAR_OUTPUT
	_rMV						:REAL;		(* Mätvärde *)
	_bLG						:BOOL; 	(*Givarfel*)
	_bDelayedLG				:BOOL;	(* Fördröjt givarfel *)
END_VAR
(* body not read: cfc101 *)
END_PROGRAM

(* POU _IOs_Uppdelat_per_skåp/HUS2_AS01/_IO/ANALOGA IN/Kort06/HUS2_AS01_Analoga_in_Kort06_AI02, FAI *)
PROGRAM HUS2_AS01_Analoga_in_Kort06_AI02
(*#####################################   Temperature Sensor Ex2   ################################################################*)
VAR
	(*===========================Configuration of terminal==========================================*)
	fbConfigureKL32xx					:FB_HVACConfigureKL32xx;
	_byCtrlKL32xx                         			AT %Q*: BYTE;
	_iDataOutKL32xx                       		AT %Q*: INT;
	_iDataInKL32xx 					AT%I*:INT;(* Raw Value from the Terminal *)
	_byStatusKL32xx 			AT%I*:BYTE;(* Statusbyte from Terminal *)

	_bScanSensor              					: BOOL;
	_tTimeOut                 					: TIME := T#5s;
	_bSetSensor               					: BOOL;
	bReady                               				: BOOL;
	byOutStatus                          			: BYTE;
	iOutDataIn                           				: INT;
	_eBusTerminalKL32xx                   		: E_HVACBusTerminal_KL32xx;
	_eStatusScanSensorType                	: E_HVACSensorType;
	_bErrorGeneral                        			: BOOL;
	_byError                              				: BYTE;
	_bErrorCommunication                  		: BOOL;
	_bErrorBusTerminalNotSupported   	: BOOL;
	_bErrorSensorType                     		: BOOL;
	_bErrorScanSensor                     		: BOOL;
	(*========================================================================================*)

	_bReset_Local					:BOOL;
	_bSetDefaultTempSens			:BOOL;

	(*========================================================================================*)
	FBHVACTemperatureSensor: FB_HVACTemperatureSensor;
	eDataSecurityType					: E_HVACDataSecurityType:=1;
	bSetDefault								:BOOL;
	iRawValue								:INT;
	byStatusRawValue						:BYTE;
	bEnableLimitCtrl							:BOOL;
	bReset									:BOOL;
	bErrorGeneral					:BOOL;
	byError							:BYTE;
	bErrorShortCircuit				:BOOL;
	bErrorBrokenSensor				:BOOL;
	bErrorHighLimit					:BOOL;
	bErrorLowLimit					:BOOL;
	bErrorCycleTime					:BOOL;
	bInvalidParameter				:BOOL;
	rOffset									:REAL;
	rHighLimit								:REAL;
	rLowLimit								:REAL;
	rReplacementValue						:REAL;
	tFilterTime								:TIME;
	eTemperatureSensorMode				:E_HVACTemperatureSensorMode:=2;
	fbAlarmD: fbDelayedAlarmMinutes;

END_VAR

VAR_INPUT
	_rKAL						: REAL;	(*Kalibrering*)
	_FT						:INT;		(*Filtertid*)
	_LG_FL					:INT;		(* Larmfördröjning givarfel *)
END_VAR

VAR_OUTPUT
	_rMV						:REAL;		(* Mätvärde *)
	_bLG						:BOOL; 	(*Givarfel*)
	_bDelayedLG				:BOOL;	(* Fördröjt givarfel *)
END_VAR
(* body not read: cfc101 *)
END_PROGRAM

(* POU _IOs_Uppdelat_per_skåp/HUS2_AS01/_IO/ANALOGA IN/Kort06/HUS2_AS01_Analoga_in_Kort06_AI06, FAI *)
PROGRAM HUS2_AS01_Analoga_in_Kort06_AI06
(*#####################################   Temperature Sensor Ex2   ################################################################*)
VAR
	(*===========================Configuration of terminal==========================================*)
	fbConfigureKL32xx					:FB_HVACConfigureKL32xx;
	_byCtrlKL32xx                         			AT %Q*: BYTE;
	_iDataOutKL32xx                       		AT %Q*: INT;
	_iDataInKL32xx 					AT%I*:INT;(* Raw Value from the Terminal *)
	_byStatusKL32xx 			AT%I*:BYTE;(* Statusbyte from Terminal *)

	_bScanSensor              					: BOOL;
	_tTimeOut                 					: TIME := T#5s;
	_bSetSensor               					: BOOL;
	bReady                               				: BOOL;
	byOutStatus                          			: BYTE;
	iOutDataIn                           				: INT;
	_eBusTerminalKL32xx                   		: E_HVACBusTerminal_KL32xx;
	_eStatusScanSensorType                	: E_HVACSensorType;
	_bErrorGeneral                        			: BOOL;
	_byError                              				: BYTE;
	_bErrorCommunication                  		: BOOL;
	_bErrorBusTerminalNotSupported   	: BOOL;
	_bErrorSensorType                     		: BOOL;
	_bErrorScanSensor                     		: BOOL;
	(*========================================================================================*)

	_bReset_Local					:BOOL;
	_bSetDefaultTempSens			:BOOL;

	(*========================================================================================*)
	FBHVACTemperatureSensor: FB_HVACTemperatureSensor;
	eDataSecurityType					: E_HVACDataSecurityType:=1;
	bSetDefault								:BOOL;
	iRawValue								:INT;
	byStatusRawValue						:BYTE;
	bEnableLimitCtrl							:BOOL;
	bReset									:BOOL;
	bErrorGeneral					:BOOL;
	byError							:BYTE;
	bErrorShortCircuit				:BOOL;
	bErrorBrokenSensor				:BOOL;
	bErrorHighLimit					:BOOL;
	bErrorLowLimit					:BOOL;
	bErrorCycleTime					:BOOL;
	bInvalidParameter				:BOOL;
	rOffset									:REAL;
	rHighLimit								:REAL;
	rLowLimit								:REAL;
	rReplacementValue						:REAL;
	tFilterTime								:TIME;
	eTemperatureSensorMode				:E_HVACTemperatureSensorMode:=2;
	fbAlarmD: fbDelayedAlarmMinutes;

END_VAR

VAR_INPUT
	_rKAL						: REAL;	(*Kalibrering*)
	_FT						:INT;		(*Filtertid*)
	_LG_FL					:INT;		(* Larmfördröjning givarfel *)
END_VAR

VAR_OUTPUT
	_rMV						:REAL;		(* Mätvärde *)
	_bLG						:BOOL; 	(*Givarfel*)
	_bDelayedLG				:BOOL;	(* Fördröjt givarfel *)
END_VAR
(* body not read: cfc101 *)
END_PROGRAM

(* POU _IOs_Uppdelat_per_skåp/HUS2_AS01/_IO/ANALOGA IN/Kort06/HUS2_AS01_Analoga_in_Kort06_AI03, FAI *)
PROGRAM HUS2_AS01_Analoga_in_Kort06_AI03
(*#####################################   Temperature Sensor Ex2   ################################################################*)
VAR
	(*===========================Configuration of terminal==========================================*)
	fbConfigureKL32xx					:FB_HVACConfigureKL32xx;
	_byCtrlKL32xx                         			AT %Q*: BYTE;
	_iDataOutKL32xx                       		AT %Q*: INT;
	_iDataInKL32xx 					AT%I*:INT;(* Raw Value from the Terminal *)
	_byStatusKL32xx 			AT%I*:BYTE;(* Statusbyte from Terminal *)

	_bScanSensor              					: BOOL;
	_tTimeOut                 					: TIME := T#5s;
	_bSetSensor               					: BOOL;
	bReady                               				: BOOL;
	byOutStatus                          			: BYTE;
	iOutDataIn                           				: INT;
	_eBusTerminalKL32xx                   		: E_HVACBusTerminal_KL32xx;
	_eStatusScanSensorType                	: E_HVACSensorType;
	_bErrorGeneral                        			: BOOL;
	_byError                              				: BYTE;
	_bErrorCommunication                  		: BOOL;
	_bErrorBusTerminalNotSupported   	: BOOL;
	_bErrorSensorType                     		: BOOL;
	_bErrorScanSensor                     		: BOOL;
	(*========================================================================================*)

	_bReset_Local					:BOOL;
	_bSetDefaultTempSens			:BOOL;

	(*========================================================================================*)
	FBHVACTemperatureSensor: FB_HVACTemperatureSensor;
	eDataSecurityType					: E_HVACDataSecurityType:=1;
	bSetDefault								:BOOL;
	iRawValue								:INT;
	byStatusRawValue						:BYTE;
	bEnableLimitCtrl							:BOOL;
	bReset									:BOOL;
	bErrorGeneral					:BOOL;
	byError							:BYTE;
	bErrorShortCircuit				:BOOL;
	bErrorBrokenSensor				:BOOL;
	bErrorHighLimit					:BOOL;
	bErrorLowLimit					:BOOL;
	bErrorCycleTime					:BOOL;
	bInvalidParameter				:BOOL;
	rOffset									:REAL;
	rHighLimit								:REAL;
	rLowLimit								:REAL;
	rReplacementValue						:REAL;
	tFilterTime								:TIME;
	eTemperatureSensorMode				:E_HVACTemperatureSensorMode:=2;
	fbAlarmD: fbDelayedAlarmMinutes;

END_VAR

VAR_INPUT
	_rKAL						: REAL;	(*Kalibrering*)
	_FT						:INT;		(*Filtertid*)
	_LG_FL					:INT;		(* Larmfördröjning givarfel *)
END_VAR

VAR_OUTPUT
	_rMV						:REAL;		(* Mätvärde *)
	_bLG						:BOOL; 	(*Givarfel*)
	_bDelayedLG				:BOOL;	(* Fördröjt givarfel *)
END_VAR
(* body not read: cfc101 *)
END_PROGRAM

(* POU _IOs_Uppdelat_per_skåp/HUS2_AS01/_IO/ANALOGA IN/Kort06/HUS2_AS01_Analoga_in_Kort06_AI07, FAI *)
PROGRAM HUS2_AS01_Analoga_in_Kort06_AI07
(*#####################################   Temperature Sensor Ex2   ################################################################*)
VAR
	(*===========================Configuration of terminal==========================================*)
	fbConfigureKL32xx					:FB_HVACConfigureKL32xx;
	_byCtrlKL32xx                         			AT %Q*: BYTE;
	_iDataOutKL32xx                       		AT %Q*: INT;
	_iDataInKL32xx 					AT%I*:INT;(* Raw Value from the Terminal *)
	_byStatusKL32xx 			AT%I*:BYTE;(* Statusbyte from Terminal *)

	_bScanSensor              					: BOOL;
	_tTimeOut                 					: TIME := T#5s;
	_bSetSensor               					: BOOL;
	bReady                               				: BOOL;
	byOutStatus                          			: BYTE;
	iOutDataIn                           				: INT;
	_eBusTerminalKL32xx                   		: E_HVACBusTerminal_KL32xx;
	_eStatusScanSensorType                	: E_HVACSensorType;
	_bErrorGeneral                        			: BOOL;
	_byError                              				: BYTE;
	_bErrorCommunication                  		: BOOL;
	_bErrorBusTerminalNotSupported   	: BOOL;
	_bErrorSensorType                     		: BOOL;
	_bErrorScanSensor                     		: BOOL;
	(*========================================================================================*)

	_bReset_Local					:BOOL;
	_bSetDefaultTempSens			:BOOL;

	(*========================================================================================*)
	FBHVACTemperatureSensor: FB_HVACTemperatureSensor;
	eDataSecurityType					: E_HVACDataSecurityType:=1;
	bSetDefault								:BOOL;
	iRawValue								:INT;
	byStatusRawValue						:BYTE;
	bEnableLimitCtrl							:BOOL;
	bReset									:BOOL;
	bErrorGeneral					:BOOL;
	byError							:BYTE;
	bErrorShortCircuit				:BOOL;
	bErrorBrokenSensor				:BOOL;
	bErrorHighLimit					:BOOL;
	bErrorLowLimit					:BOOL;
	bErrorCycleTime					:BOOL;
	bInvalidParameter				:BOOL;
	rOffset									:REAL;
	rHighLimit								:REAL;
	rLowLimit								:REAL;
	rReplacementValue						:REAL;
	tFilterTime								:TIME;
	eTemperatureSensorMode				:E_HVACTemperatureSensorMode:=2;
	fbAlarmD: fbDelayedAlarmMinutes;

END_VAR

VAR_INPUT
	_rKAL						: REAL;	(*Kalibrering*)
	_FT						:INT;		(*Filtertid*)
	_LG_FL					:INT;		(* Larmfördröjning givarfel *)
END_VAR

VAR_OUTPUT
	_rMV						:REAL;		(* Mätvärde *)
	_bLG						:BOOL; 	(*Givarfel*)
	_bDelayedLG				:BOOL;	(* Fördröjt givarfel *)
END_VAR
(* body not read: cfc101 *)
END_PROGRAM

(* POU _IOs_Uppdelat_per_skåp/HUS2_AS01/_IO/ANALOGA IN/Kort06/HUS2_AS01_Analoga_in_Kort06_AI04, FAI *)
PROGRAM HUS2_AS01_Analoga_in_Kort06_AI04
(*#####################################   Temperature Sensor Ex2   ################################################################*)
VAR
	(*===========================Configuration of terminal==========================================*)
	fbConfigureKL32xx					:FB_HVACConfigureKL32xx;
	_byCtrlKL32xx                         			AT %Q*: BYTE;
	_iDataOutKL32xx                       		AT %Q*: INT;
	_iDataInKL32xx 					AT%I*:INT;(* Raw Value from the Terminal *)
	_byStatusKL32xx 			AT%I*:BYTE;(* Statusbyte from Terminal *)

	_bScanSensor              					: BOOL;
	_tTimeOut                 					: TIME := T#5s;
	_bSetSensor               					: BOOL;
	bReady                               				: BOOL;
	byOutStatus                          			: BYTE;
	iOutDataIn                           				: INT;
	_eBusTerminalKL32xx                   		: E_HVACBusTerminal_KL32xx;
	_eStatusScanSensorType                	: E_HVACSensorType;
	_bErrorGeneral                        			: BOOL;
	_byError                              				: BYTE;
	_bErrorCommunication                  		: BOOL;
	_bErrorBusTerminalNotSupported   	: BOOL;
	_bErrorSensorType                     		: BOOL;
	_bErrorScanSensor                     		: BOOL;
	(*========================================================================================*)

	_bReset_Local					:BOOL;
	_bSetDefaultTempSens			:BOOL;

	(*========================================================================================*)
	FBHVACTemperatureSensor: FB_HVACTemperatureSensor;
	eDataSecurityType					: E_HVACDataSecurityType:=1;
	bSetDefault								:BOOL;
	iRawValue								:INT;
	byStatusRawValue						:BYTE;
	bEnableLimitCtrl							:BOOL;
	bReset									:BOOL;
	bErrorGeneral					:BOOL;
	byError							:BYTE;
	bErrorShortCircuit				:BOOL;
	bErrorBrokenSensor				:BOOL;
	bErrorHighLimit					:BOOL;
	bErrorLowLimit					:BOOL;
	bErrorCycleTime					:BOOL;
	bInvalidParameter				:BOOL;
	rOffset									:REAL;
	rHighLimit								:REAL;
	rLowLimit								:REAL;
	rReplacementValue						:REAL;
	tFilterTime								:TIME;
	eTemperatureSensorMode				:E_HVACTemperatureSensorMode:=2;
	fbAlarmD: fbDelayedAlarmMinutes;

END_VAR

VAR_INPUT
	_rKAL						: REAL;	(*Kalibrering*)
	_FT						:INT;		(*Filtertid*)
	_LG_FL					:INT;		(* Larmfördröjning givarfel *)
END_VAR

VAR_OUTPUT
	_rMV						:REAL;		(* Mätvärde *)
	_bLG						:BOOL; 	(*Givarfel*)
	_bDelayedLG				:BOOL;	(* Fördröjt givarfel *)
END_VAR
(* body not read: cfc101 *)
END_PROGRAM

(* POU _IOs_Uppdelat_per_skåp/HUS2_AS01/_IO/ANALOGA IN/Kort06/HUS2_AS01_Analoga_in_Kort06_AI08, FAI *)
PROGRAM HUS2_AS01_Analoga_in_Kort06_AI08
(*#####################################   Temperature Sensor Ex2   ################################################################*)
VAR
	(*===========================Configuration of terminal==========================================*)
	fbConfigureKL32xx					:FB_HVACConfigureKL32xx;
	_byCtrlKL32xx                         			AT %Q*: BYTE;
	_iDataOutKL32xx                       		AT %Q*: INT;
	_iDataInKL32xx 					AT%I*:INT;(* Raw Value from the Terminal *)
	_byStatusKL32xx 			AT%I*:BYTE;(* Statusbyte from Terminal *)

	_bScanSensor              					: BOOL;
	_tTimeOut                 					: TIME := T#5s;
	_bSetSensor               					: BOOL;
	bReady                               				: BOOL;
	byOutStatus                          			: BYTE;
	iOutDataIn                           				: INT;
	_eBusTerminalKL32xx                   		: E_HVACBusTerminal_KL32xx;
	_eStatusScanSensorType                	: E_HVACSensorType;
	_bErrorGeneral                        			: BOOL;
	_byError                              				: BYTE;
	_bErrorCommunication                  		: BOOL;
	_bErrorBusTerminalNotSupported   	: BOOL;
	_bErrorSensorType                     		: BOOL;
	_bErrorScanSensor                     		: BOOL;
	(*========================================================================================*)

	_bReset_Local					:BOOL;
	_bSetDefaultTempSens			:BOOL;

	(*========================================================================================*)
	FBHVACTemperatureSensor: FB_HVACTemperatureSensor;
	eDataSecurityType					: E_HVACDataSecurityType:=1;
	bSetDefault								:BOOL;
	iRawValue								:INT;
	byStatusRawValue						:BYTE;
	bEnableLimitCtrl							:BOOL;
	bReset									:BOOL;
	bErrorGeneral					:BOOL;
	byError							:BYTE;
	bErrorShortCircuit				:BOOL;
	bErrorBrokenSensor				:BOOL;
	bErrorHighLimit					:BOOL;
	bErrorLowLimit					:BOOL;
	bErrorCycleTime					:BOOL;
	bInvalidParameter				:BOOL;
	rOffset									:REAL;
	rHighLimit								:REAL;
	rLowLimit								:REAL;
	rReplacementValue						:REAL;
	tFilterTime								:TIME;
	eTemperatureSensorMode				:E_HVACTemperatureSensorMode:=2;
	fbAlarmD: fbDelayedAlarmMinutes;

END_VAR

VAR_INPUT
	_rKAL						: REAL;	(*Kalibrering*)
	_FT						:INT;		(*Filtertid*)
	_LG_FL					:INT;		(* Larmfördröjning givarfel *)
END_VAR

VAR_OUTPUT
	_rMV						:REAL;		(* Mätvärde *)
	_bLG						:BOOL; 	(*Givarfel*)
	_bDelayedLG				:BOOL;	(* Fördröjt givarfel *)
END_VAR
(* body not read: cfc101 *)
END_PROGRAM

(* POU _IOs_Uppdelat_per_skåp/HUS2_AS01/_IO/ANALOGA IN/Kort07/HUS2_AS01_Analoga_in_Kort07, CFC *)
PROGRAM HUS2_AS01_Analoga_in_Kort07
VAR
	bLG01: BOOL;
	bLG02: BOOL;
	bLG03: BOOL;
	bLG04: BOOL;
	bLG05: BOOL;
	bLG06: BOOL;
	bLG07: BOOL;
	bLG08: BOOL;

(*TEMP*)
	FT1:INT;
	LG_FL1:INT;
	FT2:INT;
	LG_FL2:INT;
	FT3:INT;
	LG_FL3:INT;
	FT4:INT;
	LG_FL4:INT;
	FT5:INT;
	LG_FL5:INT;
	FT6:INT;
	LG_FL6:INT;
	FT7:INT;
	LG_FL7:INT;
	FT8:INT;
	LG_FL8:INT;

END_VAR
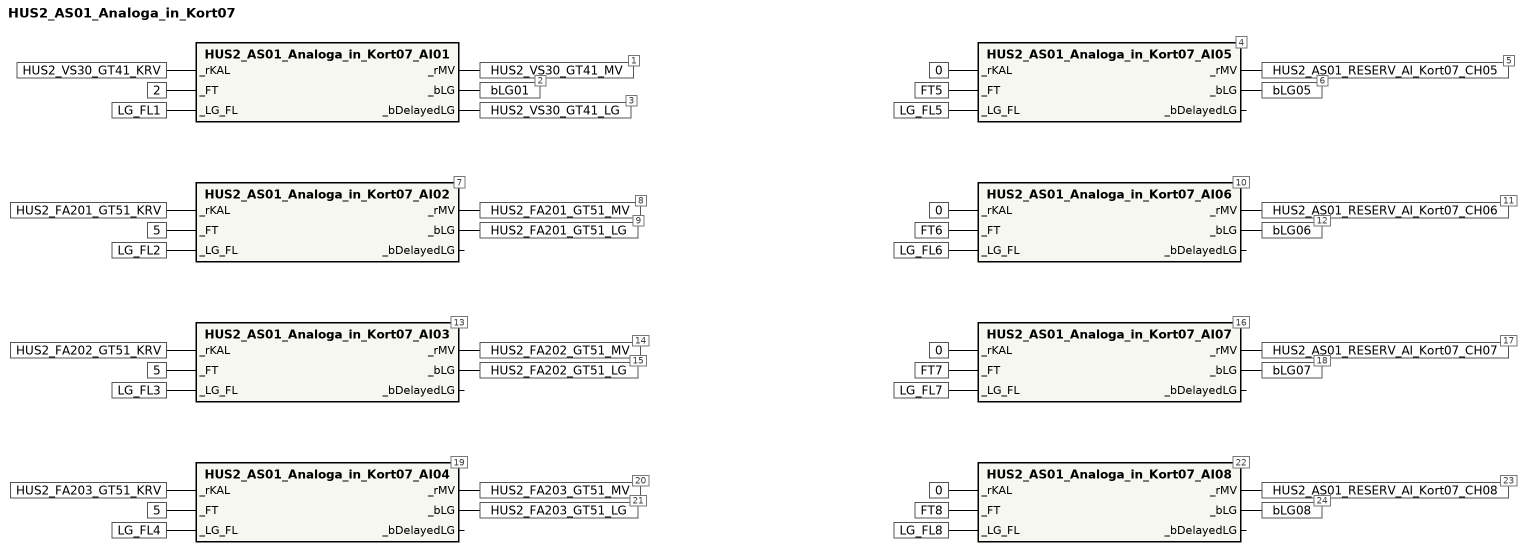
_CFC_ (* Continuous Function Chart, elements in execution order *)
#0 HUS2_AS01_Analoga_in_Kort07_AI01(_rKAL: HUS2_VS30_GT41_KRV, _FT: 2, _LG_FL: LG_FL1)
#1 HUS2_VS30_GT41_MV <= #0._rMV
#2 bLG01 <= #0._bLG
#3 HUS2_VS30_GT41_LG <= #0._bDelayedLG
#4 HUS2_AS01_Analoga_in_Kort07_AI05(_rKAL: 0, _FT: FT5, _LG_FL: LG_FL5)
#5 HUS2_AS01_RESERV_AI_Kort07_CH05 <= #4._rMV
#6 bLG05 <= #4._bLG
#7 HUS2_AS01_Analoga_in_Kort07_AI02(_rKAL: HUS2_FA201_GT51_KRV, _FT: 5, _LG_FL: LG_FL2)
#8 HUS2_FA201_GT51_MV <= #7._rMV
#9 HUS2_FA201_GT51_LG <= #7._bLG
#10 HUS2_AS01_Analoga_in_Kort07_AI06(_rKAL: 0, _FT: FT6, _LG_FL: LG_FL6)
#11 HUS2_AS01_RESERV_AI_Kort07_CH06 <= #10._rMV
#12 bLG06 <= #10._bLG
#13 HUS2_AS01_Analoga_in_Kort07_AI03(_rKAL: HUS2_FA202_GT51_KRV, _FT: 5, _LG_FL: LG_FL3)
#14 HUS2_FA202_GT51_MV <= #13._rMV
#15 HUS2_FA202_GT51_LG <= #13._bLG
#16 HUS2_AS01_Analoga_in_Kort07_AI07(_rKAL: 0, _FT: FT7, _LG_FL: LG_FL7)
#17 HUS2_AS01_RESERV_AI_Kort07_CH07 <= #16._rMV
#18 bLG07 <= #16._bLG
#19 HUS2_AS01_Analoga_in_Kort07_AI04(_rKAL: HUS2_FA203_GT51_KRV, _FT: 5, _LG_FL: LG_FL4)
#20 HUS2_FA203_GT51_MV <= #19._rMV
#21 HUS2_FA203_GT51_LG <= #19._bLG
#22 HUS2_AS01_Analoga_in_Kort07_AI08(_rKAL: 0, _FT: FT8, _LG_FL: LG_FL8)
#23 HUS2_AS01_RESERV_AI_Kort07_CH08 <= #22._rMV
#24 bLG08 <= #22._bLG
_END_CFC_
(* the same logic as Structured Text *)
HUS2_AS01_Analoga_in_Kort07_AI01(_rKAL := HUS2_VS30_GT41_KRV, _FT := 2, _LG_FL := LG_FL1);
HUS2_VS30_GT41_MV := HUS2_AS01_Analoga_in_Kort07_AI01._rMV;
bLG01 := HUS2_AS01_Analoga_in_Kort07_AI01._bLG;
HUS2_VS30_GT41_LG := HUS2_AS01_Analoga_in_Kort07_AI01._bDelayedLG;
HUS2_AS01_Analoga_in_Kort07_AI05(_rKAL := 0, _FT := FT5, _LG_FL := LG_FL5);
HUS2_AS01_RESERV_AI_Kort07_CH05 := HUS2_AS01_Analoga_in_Kort07_AI05._rMV;
bLG05 := HUS2_AS01_Analoga_in_Kort07_AI05._bLG;
HUS2_AS01_Analoga_in_Kort07_AI02(_rKAL := HUS2_FA201_GT51_KRV, _FT := 5, _LG_FL := LG_FL2);
HUS2_FA201_GT51_MV := HUS2_AS01_Analoga_in_Kort07_AI02._rMV;
HUS2_FA201_GT51_LG := HUS2_AS01_Analoga_in_Kort07_AI02._bLG;
HUS2_AS01_Analoga_in_Kort07_AI06(_rKAL := 0, _FT := FT6, _LG_FL := LG_FL6);
HUS2_AS01_RESERV_AI_Kort07_CH06 := HUS2_AS01_Analoga_in_Kort07_AI06._rMV;
bLG06 := HUS2_AS01_Analoga_in_Kort07_AI06._bLG;
HUS2_AS01_Analoga_in_Kort07_AI03(_rKAL := HUS2_FA202_GT51_KRV, _FT := 5, _LG_FL := LG_FL3);
HUS2_FA202_GT51_MV := HUS2_AS01_Analoga_in_Kort07_AI03._rMV;
HUS2_FA202_GT51_LG := HUS2_AS01_Analoga_in_Kort07_AI03._bLG;
HUS2_AS01_Analoga_in_Kort07_AI07(_rKAL := 0, _FT := FT7, _LG_FL := LG_FL7);
HUS2_AS01_RESERV_AI_Kort07_CH07 := HUS2_AS01_Analoga_in_Kort07_AI07._rMV;
bLG07 := HUS2_AS01_Analoga_in_Kort07_AI07._bLG;
HUS2_AS01_Analoga_in_Kort07_AI04(_rKAL := HUS2_FA203_GT51_KRV, _FT := 5, _LG_FL := LG_FL4);
HUS2_FA203_GT51_MV := HUS2_AS01_Analoga_in_Kort07_AI04._rMV;
HUS2_FA203_GT51_LG := HUS2_AS01_Analoga_in_Kort07_AI04._bLG;
HUS2_AS01_Analoga_in_Kort07_AI08(_rKAL := 0, _FT := FT8, _LG_FL := LG_FL8);
HUS2_AS01_RESERV_AI_Kort07_CH08 := HUS2_AS01_Analoga_in_Kort07_AI08._rMV;
bLG08 := HUS2_AS01_Analoga_in_Kort07_AI08._bLG;
END_PROGRAM

(* POU _IOs_Uppdelat_per_skåp/HUS2_AS01/_IO/ANALOGA IN/Kort07/HUS2_AS01_Analoga_in_Kort07_AI01, FAI *)
PROGRAM HUS2_AS01_Analoga_in_Kort07_AI01
(*#####################################   Temperature Sensor Ex2   ################################################################*)
VAR
	(*===========================Configuration of terminal==========================================*)
	fbConfigureKL32xx					:FB_HVACConfigureKL32xx;
	_byCtrlKL32xx                         			AT %Q*: BYTE;
	_iDataOutKL32xx                       		AT %Q*: INT;
	_iDataInKL32xx 					AT%I*:INT;(* Raw Value from the Terminal *)
	_byStatusKL32xx 			AT%I*:BYTE;(* Statusbyte from Terminal *)

	_bScanSensor              					: BOOL;
	_tTimeOut                 					: TIME := T#5s;
	_bSetSensor               					: BOOL;
	bReady                               				: BOOL;
	byOutStatus                          			: BYTE;
	iOutDataIn                           				: INT;
	_eBusTerminalKL32xx                   		: E_HVACBusTerminal_KL32xx;
	_eStatusScanSensorType                	: E_HVACSensorType;
	_bErrorGeneral                        			: BOOL;
	_byError                              				: BYTE;
	_bErrorCommunication                  		: BOOL;
	_bErrorBusTerminalNotSupported   	: BOOL;
	_bErrorSensorType                     		: BOOL;
	_bErrorScanSensor                     		: BOOL;
	(*========================================================================================*)

	_bReset_Local					:BOOL;
	_bSetDefaultTempSens			:BOOL;

	(*========================================================================================*)
	FBHVACTemperatureSensor: FB_HVACTemperatureSensor;
	eDataSecurityType					: E_HVACDataSecurityType:=1;
	bSetDefault								:BOOL;
	iRawValue								:INT;
	byStatusRawValue						:BYTE;
	bEnableLimitCtrl							:BOOL;
	bReset									:BOOL;
	bErrorGeneral					:BOOL;
	byError							:BYTE;
	bErrorShortCircuit				:BOOL;
	bErrorBrokenSensor				:BOOL;
	bErrorHighLimit					:BOOL;
	bErrorLowLimit					:BOOL;
	bErrorCycleTime					:BOOL;
	bInvalidParameter				:BOOL;
	rOffset									:REAL;
	rHighLimit								:REAL;
	rLowLimit								:REAL;
	rReplacementValue						:REAL;
	tFilterTime								:TIME;
	eTemperatureSensorMode				:E_HVACTemperatureSensorMode:=2;
	fbAlarmD: fbDelayedAlarmMinutes;

END_VAR

VAR_INPUT
	_rKAL						: REAL;	(*Kalibrering*)
	_FT						:INT;		(*Filtertid*)
	_LG_FL					:INT;		(* Larmfördröjning givarfel *)
END_VAR

VAR_OUTPUT
	_rMV						:REAL;		(* Mätvärde *)
	_bLG						:BOOL; 	(*Givarfel*)
	_bDelayedLG				:BOOL;	(* Fördröjt givarfel *)
END_VAR
(* body not read: cfc101 *)
END_PROGRAM

(* POU _IOs_Uppdelat_per_skåp/HUS2_AS01/_IO/ANALOGA IN/Kort07/HUS2_AS01_Analoga_in_Kort07_AI05, FAI *)
PROGRAM HUS2_AS01_Analoga_in_Kort07_AI05
(*#####################################   Temperature Sensor Ex2   ################################################################*)
VAR
	(*===========================Configuration of terminal==========================================*)
	fbConfigureKL32xx					:FB_HVACConfigureKL32xx;
	_byCtrlKL32xx                         			AT %Q*: BYTE;
	_iDataOutKL32xx                       		AT %Q*: INT;
	_iDataInKL32xx 					AT%I*:INT;(* Raw Value from the Terminal *)
	_byStatusKL32xx 			AT%I*:BYTE;(* Statusbyte from Terminal *)

	_bScanSensor              					: BOOL;
	_tTimeOut                 					: TIME := T#5s;
	_bSetSensor               					: BOOL;
	bReady                               				: BOOL;
	byOutStatus                          			: BYTE;
	iOutDataIn                           				: INT;
	_eBusTerminalKL32xx                   		: E_HVACBusTerminal_KL32xx;
	_eStatusScanSensorType                	: E_HVACSensorType;
	_bErrorGeneral                        			: BOOL;
	_byError                              				: BYTE;
	_bErrorCommunication                  		: BOOL;
	_bErrorBusTerminalNotSupported   	: BOOL;
	_bErrorSensorType                     		: BOOL;
	_bErrorScanSensor                     		: BOOL;
	(*========================================================================================*)

	_bReset_Local					:BOOL;
	_bSetDefaultTempSens			:BOOL;

	(*========================================================================================*)
	FBHVACTemperatureSensor: FB_HVACTemperatureSensor;
	eDataSecurityType					: E_HVACDataSecurityType:=1;
	bSetDefault								:BOOL;
	iRawValue								:INT;
	byStatusRawValue						:BYTE;
	bEnableLimitCtrl							:BOOL;
	bReset									:BOOL;
	bErrorGeneral					:BOOL;
	byError							:BYTE;
	bErrorShortCircuit				:BOOL;
	bErrorBrokenSensor				:BOOL;
	bErrorHighLimit					:BOOL;
	bErrorLowLimit					:BOOL;
	bErrorCycleTime					:BOOL;
	bInvalidParameter				:BOOL;
	rOffset									:REAL;
	rHighLimit								:REAL;
	rLowLimit								:REAL;
	rReplacementValue						:REAL;
	tFilterTime								:TIME;
	eTemperatureSensorMode				:E_HVACTemperatureSensorMode:=2;
	fbAlarmD: fbDelayedAlarmMinutes;

END_VAR

VAR_INPUT
	_rKAL						: REAL;	(*Kalibrering*)
	_FT						:INT;		(*Filtertid*)
	_LG_FL					:INT;		(* Larmfördröjning givarfel *)
END_VAR

VAR_OUTPUT
	_rMV						:REAL;		(* Mätvärde *)
	_bLG						:BOOL; 	(*Givarfel*)
	_bDelayedLG				:BOOL;	(* Fördröjt givarfel *)
END_VAR
(* body not read: cfc101 *)
END_PROGRAM

(* POU _IOs_Uppdelat_per_skåp/HUS2_AS01/_IO/ANALOGA IN/Kort07/HUS2_AS01_Analoga_in_Kort07_AI02, FAI *)
PROGRAM HUS2_AS01_Analoga_in_Kort07_AI02
(*#####################################   Temperature Sensor Ex2   ################################################################*)
VAR
	(*===========================Configuration of terminal==========================================*)
	fbConfigureKL32xx					:FB_HVACConfigureKL32xx;
	_byCtrlKL32xx                         			AT %Q*: BYTE;
	_iDataOutKL32xx                       		AT %Q*: INT;
	_iDataInKL32xx 					AT%I*:INT;(* Raw Value from the Terminal *)
	_byStatusKL32xx 			AT%I*:BYTE;(* Statusbyte from Terminal *)

	_bScanSensor              					: BOOL;
	_tTimeOut                 					: TIME := T#5s;
	_bSetSensor               					: BOOL;
	bReady                               				: BOOL;
	byOutStatus                          			: BYTE;
	iOutDataIn                           				: INT;
	_eBusTerminalKL32xx                   		: E_HVACBusTerminal_KL32xx;
	_eStatusScanSensorType                	: E_HVACSensorType;
	_bErrorGeneral                        			: BOOL;
	_byError                              				: BYTE;
	_bErrorCommunication                  		: BOOL;
	_bErrorBusTerminalNotSupported   	: BOOL;
	_bErrorSensorType                     		: BOOL;
	_bErrorScanSensor                     		: BOOL;
	(*========================================================================================*)

	_bReset_Local					:BOOL;
	_bSetDefaultTempSens			:BOOL;

	(*========================================================================================*)
	FBHVACTemperatureSensor: FB_HVACTemperatureSensor;
	eDataSecurityType					: E_HVACDataSecurityType:=1;
	bSetDefault								:BOOL;
	iRawValue								:INT;
	byStatusRawValue						:BYTE;
	bEnableLimitCtrl							:BOOL;
	bReset									:BOOL;
	bErrorGeneral					:BOOL;
	byError							:BYTE;
	bErrorShortCircuit				:BOOL;
	bErrorBrokenSensor				:BOOL;
	bErrorHighLimit					:BOOL;
	bErrorLowLimit					:BOOL;
	bErrorCycleTime					:BOOL;
	bInvalidParameter				:BOOL;
	rOffset									:REAL;
	rHighLimit								:REAL;
	rLowLimit								:REAL;
	rReplacementValue						:REAL;
	tFilterTime								:TIME;
	eTemperatureSensorMode				:E_HVACTemperatureSensorMode:=2;
	fbAlarmD: fbDelayedAlarmMinutes;

END_VAR

VAR_INPUT
	_rKAL						: REAL;	(*Kalibrering*)
	_FT						:INT;		(*Filtertid*)
	_LG_FL					:INT;		(* Larmfördröjning givarfel *)
END_VAR

VAR_OUTPUT
	_rMV						:REAL;		(* Mätvärde *)
	_bLG						:BOOL; 	(*Givarfel*)
	_bDelayedLG				:BOOL;	(* Fördröjt givarfel *)
END_VAR
(* body not read: cfc101 *)
END_PROGRAM

(* POU _IOs_Uppdelat_per_skåp/HUS2_AS01/_IO/ANALOGA IN/Kort07/HUS2_AS01_Analoga_in_Kort07_AI06, FAI *)
PROGRAM HUS2_AS01_Analoga_in_Kort07_AI06
(*#####################################   Temperature Sensor Ex2   ################################################################*)
VAR
	(*===========================Configuration of terminal==========================================*)
	fbConfigureKL32xx					:FB_HVACConfigureKL32xx;
	_byCtrlKL32xx                         			AT %Q*: BYTE;
	_iDataOutKL32xx                       		AT %Q*: INT;
	_iDataInKL32xx 					AT%I*:INT;(* Raw Value from the Terminal *)
	_byStatusKL32xx 			AT%I*:BYTE;(* Statusbyte from Terminal *)

	_bScanSensor              					: BOOL;
	_tTimeOut                 					: TIME := T#5s;
	_bSetSensor               					: BOOL;
	bReady                               				: BOOL;
	byOutStatus                          			: BYTE;
	iOutDataIn                           				: INT;
	_eBusTerminalKL32xx                   		: E_HVACBusTerminal_KL32xx;
	_eStatusScanSensorType                	: E_HVACSensorType;
	_bErrorGeneral                        			: BOOL;
	_byError                              				: BYTE;
	_bErrorCommunication                  		: BOOL;
	_bErrorBusTerminalNotSupported   	: BOOL;
	_bErrorSensorType                     		: BOOL;
	_bErrorScanSensor                     		: BOOL;
	(*========================================================================================*)

	_bReset_Local					:BOOL;
	_bSetDefaultTempSens			:BOOL;

	(*========================================================================================*)
	FBHVACTemperatureSensor: FB_HVACTemperatureSensor;
	eDataSecurityType					: E_HVACDataSecurityType:=1;
	bSetDefault								:BOOL;
	iRawValue								:INT;
	byStatusRawValue						:BYTE;
	bEnableLimitCtrl							:BOOL;
	bReset									:BOOL;
	bErrorGeneral					:BOOL;
	byError							:BYTE;
	bErrorShortCircuit				:BOOL;
	bErrorBrokenSensor				:BOOL;
	bErrorHighLimit					:BOOL;
	bErrorLowLimit					:BOOL;
	bErrorCycleTime					:BOOL;
	bInvalidParameter				:BOOL;
	rOffset									:REAL;
	rHighLimit								:REAL;
	rLowLimit								:REAL;
	rReplacementValue						:REAL;
	tFilterTime								:TIME;
	eTemperatureSensorMode				:E_HVACTemperatureSensorMode:=2;
	fbAlarmD: fbDelayedAlarmMinutes;

END_VAR

VAR_INPUT
	_rKAL						: REAL;	(*Kalibrering*)
	_FT						:INT;		(*Filtertid*)
	_LG_FL					:INT;		(* Larmfördröjning givarfel *)
END_VAR

VAR_OUTPUT
	_rMV						:REAL;		(* Mätvärde *)
	_bLG						:BOOL; 	(*Givarfel*)
	_bDelayedLG				:BOOL;	(* Fördröjt givarfel *)
END_VAR
(* body not read: cfc101 *)
END_PROGRAM

(* POU _IOs_Uppdelat_per_skåp/HUS2_AS01/_IO/ANALOGA IN/Kort07/HUS2_AS01_Analoga_in_Kort07_AI03, FAI *)
PROGRAM HUS2_AS01_Analoga_in_Kort07_AI03
(*#####################################   Temperature Sensor Ex2   ################################################################*)
VAR
	(*===========================Configuration of terminal==========================================*)
	fbConfigureKL32xx					:FB_HVACConfigureKL32xx;
	_byCtrlKL32xx                         			AT %Q*: BYTE;
	_iDataOutKL32xx                       		AT %Q*: INT;
	_iDataInKL32xx 					AT%I*:INT;(* Raw Value from the Terminal *)
	_byStatusKL32xx 			AT%I*:BYTE;(* Statusbyte from Terminal *)

	_bScanSensor              					: BOOL;
	_tTimeOut                 					: TIME := T#5s;
	_bSetSensor               					: BOOL;
	bReady                               				: BOOL;
	byOutStatus                          			: BYTE;
	iOutDataIn                           				: INT;
	_eBusTerminalKL32xx                   		: E_HVACBusTerminal_KL32xx;
	_eStatusScanSensorType                	: E_HVACSensorType;
	_bErrorGeneral                        			: BOOL;
	_byError                              				: BYTE;
	_bErrorCommunication                  		: BOOL;
	_bErrorBusTerminalNotSupported   	: BOOL;
	_bErrorSensorType                     		: BOOL;
	_bErrorScanSensor                     		: BOOL;
	(*========================================================================================*)

	_bReset_Local					:BOOL;
	_bSetDefaultTempSens			:BOOL;

	(*========================================================================================*)
	FBHVACTemperatureSensor: FB_HVACTemperatureSensor;
	eDataSecurityType					: E_HVACDataSecurityType:=1;
	bSetDefault								:BOOL;
	iRawValue								:INT;
	byStatusRawValue						:BYTE;
	bEnableLimitCtrl							:BOOL;
	bReset									:BOOL;
	bErrorGeneral					:BOOL;
	byError							:BYTE;
	bErrorShortCircuit				:BOOL;
	bErrorBrokenSensor				:BOOL;
	bErrorHighLimit					:BOOL;
	bErrorLowLimit					:BOOL;
	bErrorCycleTime					:BOOL;
	bInvalidParameter				:BOOL;
	rOffset									:REAL;
	rHighLimit								:REAL;
	rLowLimit								:REAL;
	rReplacementValue						:REAL;
	tFilterTime								:TIME;
	eTemperatureSensorMode				:E_HVACTemperatureSensorMode:=2;
	fbAlarmD: fbDelayedAlarmMinutes;

END_VAR

VAR_INPUT
	_rKAL						: REAL;	(*Kalibrering*)
	_FT						:INT;		(*Filtertid*)
	_LG_FL					:INT;		(* Larmfördröjning givarfel *)
END_VAR

VAR_OUTPUT
	_rMV						:REAL;		(* Mätvärde *)
	_bLG						:BOOL; 	(*Givarfel*)
	_bDelayedLG				:BOOL;	(* Fördröjt givarfel *)
END_VAR
(* body not read: cfc101 *)
END_PROGRAM

(* POU _IOs_Uppdelat_per_skåp/HUS2_AS01/_IO/ANALOGA IN/Kort07/HUS2_AS01_Analoga_in_Kort07_AI07, FAI *)
PROGRAM HUS2_AS01_Analoga_in_Kort07_AI07
(*#####################################   Temperature Sensor Ex2   ################################################################*)
VAR
	(*===========================Configuration of terminal==========================================*)
	fbConfigureKL32xx					:FB_HVACConfigureKL32xx;
	_byCtrlKL32xx                         			AT %Q*: BYTE;
	_iDataOutKL32xx                       		AT %Q*: INT;
	_iDataInKL32xx 					AT%I*:INT;(* Raw Value from the Terminal *)
	_byStatusKL32xx 			AT%I*:BYTE;(* Statusbyte from Terminal *)

	_bScanSensor              					: BOOL;
	_tTimeOut                 					: TIME := T#5s;
	_bSetSensor               					: BOOL;
	bReady                               				: BOOL;
	byOutStatus                          			: BYTE;
	iOutDataIn                           				: INT;
	_eBusTerminalKL32xx                   		: E_HVACBusTerminal_KL32xx;
	_eStatusScanSensorType                	: E_HVACSensorType;
	_bErrorGeneral                        			: BOOL;
	_byError                              				: BYTE;
	_bErrorCommunication                  		: BOOL;
	_bErrorBusTerminalNotSupported   	: BOOL;
	_bErrorSensorType                     		: BOOL;
	_bErrorScanSensor                     		: BOOL;
	(*========================================================================================*)

	_bReset_Local					:BOOL;
	_bSetDefaultTempSens			:BOOL;

	(*========================================================================================*)
	FBHVACTemperatureSensor: FB_HVACTemperatureSensor;
	eDataSecurityType					: E_HVACDataSecurityType:=1;
	bSetDefault								:BOOL;
	iRawValue								:INT;
	byStatusRawValue						:BYTE;
	bEnableLimitCtrl							:BOOL;
	bReset									:BOOL;
	bErrorGeneral					:BOOL;
	byError							:BYTE;
	bErrorShortCircuit				:BOOL;
	bErrorBrokenSensor				:BOOL;
	bErrorHighLimit					:BOOL;
	bErrorLowLimit					:BOOL;
	bErrorCycleTime					:BOOL;
	bInvalidParameter				:BOOL;
	rOffset									:REAL;
	rHighLimit								:REAL;
	rLowLimit								:REAL;
	rReplacementValue						:REAL;
	tFilterTime								:TIME;
	eTemperatureSensorMode				:E_HVACTemperatureSensorMode:=2;
	fbAlarmD: fbDelayedAlarmMinutes;

END_VAR

VAR_INPUT
	_rKAL						: REAL;	(*Kalibrering*)
	_FT						:INT;		(*Filtertid*)
	_LG_FL					:INT;		(* Larmfördröjning givarfel *)
END_VAR

VAR_OUTPUT
	_rMV						:REAL;		(* Mätvärde *)
	_bLG						:BOOL; 	(*Givarfel*)
	_bDelayedLG				:BOOL;	(* Fördröjt givarfel *)
END_VAR
(* body not read: cfc101 *)
END_PROGRAM

(* POU _IOs_Uppdelat_per_skåp/HUS2_AS01/_IO/ANALOGA IN/Kort07/HUS2_AS01_Analoga_in_Kort07_AI04, FAI *)
PROGRAM HUS2_AS01_Analoga_in_Kort07_AI04
(*#####################################   Temperature Sensor Ex2   ################################################################*)
VAR
	(*===========================Configuration of terminal==========================================*)
	fbConfigureKL32xx					:FB_HVACConfigureKL32xx;
	_byCtrlKL32xx                         			AT %Q*: BYTE;
	_iDataOutKL32xx                       		AT %Q*: INT;
	_iDataInKL32xx 					AT%I*:INT;(* Raw Value from the Terminal *)
	_byStatusKL32xx 			AT%I*:BYTE;(* Statusbyte from Terminal *)

	_bScanSensor              					: BOOL;
	_tTimeOut                 					: TIME := T#5s;
	_bSetSensor               					: BOOL;
	bReady                               				: BOOL;
	byOutStatus                          			: BYTE;
	iOutDataIn                           				: INT;
	_eBusTerminalKL32xx                   		: E_HVACBusTerminal_KL32xx;
	_eStatusScanSensorType                	: E_HVACSensorType;
	_bErrorGeneral                        			: BOOL;
	_byError                              				: BYTE;
	_bErrorCommunication                  		: BOOL;
	_bErrorBusTerminalNotSupported   	: BOOL;
	_bErrorSensorType                     		: BOOL;
	_bErrorScanSensor                     		: BOOL;
	(*========================================================================================*)

	_bReset_Local					:BOOL;
	_bSetDefaultTempSens			:BOOL;

	(*========================================================================================*)
	FBHVACTemperatureSensor: FB_HVACTemperatureSensor;
	eDataSecurityType					: E_HVACDataSecurityType:=1;
	bSetDefault								:BOOL;
	iRawValue								:INT;
	byStatusRawValue						:BYTE;
	bEnableLimitCtrl							:BOOL;
	bReset									:BOOL;
	bErrorGeneral					:BOOL;
	byError							:BYTE;
	bErrorShortCircuit				:BOOL;
	bErrorBrokenSensor				:BOOL;
	bErrorHighLimit					:BOOL;
	bErrorLowLimit					:BOOL;
	bErrorCycleTime					:BOOL;
	bInvalidParameter				:BOOL;
	rOffset									:REAL;
	rHighLimit								:REAL;
	rLowLimit								:REAL;
	rReplacementValue						:REAL;
	tFilterTime								:TIME;
	eTemperatureSensorMode				:E_HVACTemperatureSensorMode:=2;
	fbAlarmD: fbDelayedAlarmMinutes;

END_VAR

VAR_INPUT
	_rKAL						: REAL;	(*Kalibrering*)
	_FT						:INT;		(*Filtertid*)
	_LG_FL					:INT;		(* Larmfördröjning givarfel *)
END_VAR

VAR_OUTPUT
	_rMV						:REAL;		(* Mätvärde *)
	_bLG						:BOOL; 	(*Givarfel*)
	_bDelayedLG				:BOOL;	(* Fördröjt givarfel *)
END_VAR
(* body not read: cfc101 *)
END_PROGRAM

(* POU _IOs_Uppdelat_per_skåp/HUS2_AS01/_IO/ANALOGA IN/Kort07/HUS2_AS01_Analoga_in_Kort07_AI08, FAI *)
PROGRAM HUS2_AS01_Analoga_in_Kort07_AI08
(*#####################################   Temperature Sensor Ex2   ################################################################*)
VAR
	(*===========================Configuration of terminal==========================================*)
	fbConfigureKL32xx					:FB_HVACConfigureKL32xx;
	_byCtrlKL32xx                         			AT %Q*: BYTE;
	_iDataOutKL32xx                       		AT %Q*: INT;
	_iDataInKL32xx 					AT%I*:INT;(* Raw Value from the Terminal *)
	_byStatusKL32xx 			AT%I*:BYTE;(* Statusbyte from Terminal *)

	_bScanSensor              					: BOOL;
	_tTimeOut                 					: TIME := T#5s;
	_bSetSensor               					: BOOL;
	bReady                               				: BOOL;
	byOutStatus                          			: BYTE;
	iOutDataIn                           				: INT;
	_eBusTerminalKL32xx                   		: E_HVACBusTerminal_KL32xx;
	_eStatusScanSensorType                	: E_HVACSensorType;
	_bErrorGeneral                        			: BOOL;
	_byError                              				: BYTE;
	_bErrorCommunication                  		: BOOL;
	_bErrorBusTerminalNotSupported   	: BOOL;
	_bErrorSensorType                     		: BOOL;
	_bErrorScanSensor                     		: BOOL;
	(*========================================================================================*)

	_bReset_Local					:BOOL;
	_bSetDefaultTempSens			:BOOL;

	(*========================================================================================*)
	FBHVACTemperatureSensor: FB_HVACTemperatureSensor;
	eDataSecurityType					: E_HVACDataSecurityType:=1;
	bSetDefault								:BOOL;
	iRawValue								:INT;
	byStatusRawValue						:BYTE;
	bEnableLimitCtrl							:BOOL;
	bReset									:BOOL;
	bErrorGeneral					:BOOL;
	byError							:BYTE;
	bErrorShortCircuit				:BOOL;
	bErrorBrokenSensor				:BOOL;
	bErrorHighLimit					:BOOL;
	bErrorLowLimit					:BOOL;
	bErrorCycleTime					:BOOL;
	bInvalidParameter				:BOOL;
	rOffset									:REAL;
	rHighLimit								:REAL;
	rLowLimit								:REAL;
	rReplacementValue						:REAL;
	tFilterTime								:TIME;
	eTemperatureSensorMode				:E_HVACTemperatureSensorMode:=2;
	fbAlarmD: fbDelayedAlarmMinutes;

END_VAR

VAR_INPUT
	_rKAL						: REAL;	(*Kalibrering*)
	_FT						:INT;		(*Filtertid*)
	_LG_FL					:INT;		(* Larmfördröjning givarfel *)
END_VAR

VAR_OUTPUT
	_rMV						:REAL;		(* Mätvärde *)
	_bLG						:BOOL; 	(*Givarfel*)
	_bDelayedLG				:BOOL;	(* Fördröjt givarfel *)
END_VAR
(* body not read: cfc101 *)
END_PROGRAM

(* POU _IOs_Uppdelat_per_skåp/HUS2_AS01/_IO/ANALOGA IN/HUS2_AS01_Analoga_in_Kort08, FAI *)
PROGRAM HUS2_AS01_Analoga_in_Kort08
VAR
	fbAI1: FB_HVACAnalogInput;
	eDataSecurityType        : E_HVACDataSecurityType;
	bSetDefault              : BOOL;
	bEnableLimitCtrl         : BOOL;
	bCtrlVoltage             : BOOL;

	byState                 : BYTE;
	bError                  : BOOL;
	eErrorCode              : E_HVACErrorCodes;
	bErrorHighLimit         : BOOL;
	bErrorLowLimit          : BOOL;
	bErrorGeneral           : BOOL;
	byError                 : BYTE;
	bInvalidParameter       : BOOL;
	iHighRange       : INT;
	iLowRange        : INT;
	rHighRange       : REAL;
	rLowRange        : REAL;
	rHighLimit       : REAL;
	rLowLimit        : REAL;
	tFilterTime      : TIME;
	rOffset          : REAL;

	fbAI2: FB_HVACAnalogInput;
	bSetDefault2              : BOOL;
	bEnableLimitCtrl2         : BOOL;
	bCtrlVoltage2             : BOOL;
	byState2                 : BYTE;
	bError2                  : BOOL;
	eErrorCode2              : E_HVACErrorCodes;
	bErrorHighLimit2         : BOOL;
	bErrorLowLimit2          : BOOL;
	bErrorGeneral2           : BOOL;
	byError2                 : BYTE;
	bInvalidParameter2       : BOOL;
	iHighRange2       : INT;
	iLowRange2        : INT;
	rHighRange2       : REAL;
	rLowRange2        : REAL;
	rHighLimit2       : REAL;
	rLowLimit2        : REAL;
	tFilterTime2      : TIME;
	rOffset2          : REAL;

	fbAI3: FB_HVACAnalogInput;
	bSetDefault3              : BOOL;
	bEnableLimitCtrl3         : BOOL;
	bCtrlVoltage3             : BOOL;

	byState3                 : BYTE;
	bError3                  : BOOL;
	eErrorCode3              : E_HVACErrorCodes;
	bErrorHighLimit3         : BOOL;
	bErrorLowLimit3          : BOOL;
	bErrorGeneral3           : BOOL;
	byError3                 : BYTE;
	bInvalidParameter3       : BOOL;
	iHighRange3       : INT;
	iLowRange3        : INT;
	rHighRange3       : REAL;
	rLowRange3        : REAL;
	rHighLimit3       : REAL;
	rLowLimit3        : REAL;
	tFilterTime3      : TIME;
	rOffset3          : REAL;

	fbAI4: FB_HVACAnalogInput;
	bSetDefault4              : BOOL;
	bEnableLimitCtrl4         : BOOL;
	bCtrlVoltage4             : BOOL;
	byState4                 : BYTE;
	bError4                  : BOOL;
	eErrorCode4              : E_HVACErrorCodes;
	bErrorHighLimit4         : BOOL;
	bErrorLowLimit4          : BOOL;
	bErrorGeneral4           : BOOL;
	byError4                 : BYTE;
	bInvalidParameteR4       : BOOL;
	iHighRange4       : INT;
	iLowRange4        : INT;
	rHighRange4       : REAL;
	rLowRange4        : REAL;
	rHighLimit4       : REAL;
	rLowLimit4        : REAL;
	tFilterTime4      : TIME;
	rOffset4          : REAL;

	fbAI5: FB_HVACAnalogInput;
	bSetDefault5              : BOOL;
	bEnableLimitCtrl5         : BOOL;
	bCtrlVoltage5             : BOOL;
	byState5                 : BYTE;
	bError5                  : BOOL;
	eErrorCode5              : E_HVACErrorCodes;
	bErrorHighLimit5         : BOOL;
	bErrorLowLimit5          : BOOL;
	bErrorGeneral5           : BOOL;
	byError5                 : BYTE;
	bInvalidParameteR5       : BOOL;
	iHighRange5       : INT;
	iLowRange5        : INT;
	rHighRange5       : REAL;
	rLowRange5        : REAL;
	rHighLimit5       : REAL;
	rLowLimit5        : REAL;
	tFilterTime5      : TIME;
	rOffset5          : REAL;

	fbAI6: FB_HVACAnalogInput;
	bSetDefault6              : BOOL;
	bEnableLimitCtrl6         : BOOL;
	bCtrlVoltage6             : BOOL;
	byState6                : BYTE;
	bError6                  : BOOL;
	eErrorCode6              : E_HVACErrorCodes;
	bErrorHighLimit6         : BOOL;
	bErrorLowLimit6          : BOOL;
	bErrorGeneral6           : BOOL;
	byError6                 : BYTE;
	bInvalidParameteR6       : BOOL;
	iHighRange6       : INT;
	iLowRange6        : INT;
	rHighRange6       : REAL;
	rLowRange6        : REAL;
	rHighLimit6       : REAL;
	rLowLimit6        : REAL;
	tFilterTime6      : TIME;
	rOffset6          : REAL;

	fbAI7: FB_HVACAnalogInput;
	bSetDefault7              : BOOL;
	bEnableLimitCtrl7         : BOOL;
	bCtrlVoltage7             : BOOL;
	byState7                : BYTE;
	bError7                  : BOOL;
	eErrorCode7              : E_HVACErrorCodes;
	bErrorHighLimit7        : BOOL;
	bErrorLowLimit7          : BOOL;
	bErrorGeneral7           : BOOL;
	byError7                 : BYTE;
	bInvalidParameteR7       : BOOL;
	iHighRange7       : INT;
	iLowRange7        : INT;
	rHighRange7       : REAL;
	rLowRange7        : REAL;
	rHighLimit7       : REAL;
	rLowLimit7        : REAL;
	tFilterTime7      : TIME;
	rOffset7         : REAL;

	fbAI8: FB_HVACAnalogInput;
	bSetDefault8              : BOOL;
	bEnableLimitCtrl8         : BOOL;
	bCtrlVoltage8             : BOOL;
	byState8                : BYTE;
	bError8                  : BOOL;
	eErrorCode8              : E_HVACErrorCodes;
	bErrorHighLimit8        : BOOL;
	bErrorLowLimit8          : BOOL;
	bErrorGeneral8           : BOOL;
	byError8                 : BYTE;
	bInvalidParameteR8       : BOOL;
	iHighRange8       : INT;
	iLowRange8        : INT;
	rHighRange8       : REAL;
	rLowRange8        : REAL;
	rHighLimit8       : REAL;
	rLowLimit8        : REAL;
	tFilterTime8      : TIME;
	rOffset8         : REAL;


	fbPersistent_LLimit: FB_HVACPersistent_Real;
	fbPersistent_HLimit: FB_HVACPersistent_Real;
	fbPersistent_LLimit2: FB_HVACPersistent_Real;
	fbPersistent_HLimit2: FB_HVACPersistent_Real;
	fbPersistent_LLimit3: FB_HVACPersistent_Real;
	fbPersistent_HLimit3: FB_HVACPersistent_Real;
	fbPersistent_LLimit4: FB_HVACPersistent_Real;
	fbPersistent_HLimit4: FB_HVACPersistent_Real;
	fbPersistent_LLimit5: FB_HVACPersistent_Real;
	fbPersistent_HLimit5: FB_HVACPersistent_Real;
	fbPersistent_LLimit6: FB_HVACPersistent_Real;
	fbPersistent_HLimit6: FB_HVACPersistent_Real;
	fbPersistent_LLimit7: FB_HVACPersistent_Real;
	fbPersistent_HLimit7: FB_HVACPersistent_Real;
	fbPersistent_LLimit8: FB_HVACPersistent_Real;
	fbPersistent_HLimit8: FB_HVACPersistent_Real;
	bSetDefault_Local: BOOL;
	bReset_Local: BOOL;





END_VAR
(* body not read: cfc97 *)
END_PROGRAM

(* POU _IOs_Uppdelat_per_skåp/HUS2_AS01/_IO/ANALOGA UT/Kort08/HUS2_AS01_Analoga_ut_Kort09, CFC *)
PROGRAM HUS2_AS01_Analoga_ut_Kort09
VAR

	Conversion_AU1: fbConversionScale;
	Conversion_AU2: fbConversionScale;
	Conversion_AU3: fbConversionScale;
	Conversion_AU4: fbConversionScale;
	Conversion_AU5: fbConversionScale;
	Conversion_AU6: fbConversionScale;
	Conversion_AU7: fbConversionScale;
	Conversion_AU8: fbConversionScale;

